KUKA KRL program: MyProgram_178().src

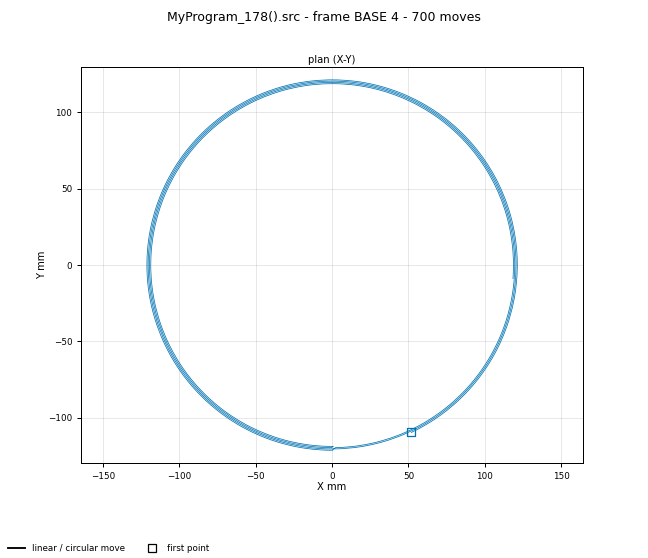
[picture p0: tool path of MyProgram_178().src in frame BASE 4, 700 of 700 moves have a stored position in this frame; points joined in program order, loops and branches not executed]
&ACCESS RVP
&REL 1
&PARAM TEMPLATE = C:\KRC\Roboter\Template\vorgabe
&PARAM EDITMASK = *
DEF MyProgram_178()
; ---- Setting reference (Base) ----
$BASE = BASE_DATA[4]

; --------------------------
; ---- Setting tool (TCP) ----
$TOOL = TOOL_DATA[3]
; --------------------------

$VEL.CP = VEL_APROX_PRINT
Startdeposition()
$VEL.CP = VEL_PRINT
LIN {X 51.9075,Y -109.6926,Z 131,A -67.6715,B 24.9586,C -1.4872,E1 25.07,E2 513.8234} C_DIS
LIN {X 55.7576,Y -107.7868,Z 131,A -65.6917,B 24.9586,C -1.4882,E1 25.0749,E2 511.8466} C_DIS
LIN {X 59.8932,Y -105.5443,Z 131,A -63.4292,B 24.9582,C -1.4942,E1 25.0805,E2 509.5764} C_DIS
LIN {X 64.6014,Y -102.7303,Z 131,A -60.7158,B 24.9576,C -1.5052,E1 25.087,E2 506.8455} C_DIS
LIN {X 68.8736,Y -99.916,Z 131,A -58.1491,B 24.9568,C -1.5177,E1 25.0929,E2 504.2581} C_DIS
LIN {X 71.8723,Y -97.7815,Z 131,A -56.8988,B 24.958,C -1.4972,E1 25.0956,E2 503.0607} C_DIS
LIN {X 75.2087,Y -95.2388,Z 131,A -54.7915,B 24.9574,C -1.5078,E1 25.1003,E2 500.9361} C_DIS
LIN {X 80.6749,Y -90.6547,Z 131,A -51.0171,B 24.9558,C -1.5358,E1 25.1084,E2 497.1104} C_DIS
LIN {X 83.659,Y -87.9089,Z 131,A -49.496,B 24.9567,C -1.5207,E1 25.1114,E2 495.631} C_DIS
LIN {X 86.4848,Y -85.1299,Z 131,A -47.1581,B 24.9551,C -1.5488,E1 25.1161,E2 493.2369} C_DIS
LIN {X 89.5631,Y -81.8851,Z 131,A -44.7373,B 24.9538,C -1.5698,E1 25.1207,E2 490.7771} C_DIS
LIN {X 93.4926,Y -77.368,Z 131,A -42.9248,B 24.9564,C -1.5263,E1 25.1238,E2 489.0757} C_DIS
LIN {X 96.0124,Y -74.2176,Z 131,A -40.5836,B 24.9548,C -1.5533,E1 25.1279,E2 486.6817} C_DIS
LIN {X 98.0547,Y -71.4981,Z 131,A -38.8834,B 24.9543,C -1.5625,E1 25.1307,E2 484.9679} C_DIS
LIN {X 100.3111,Y -68.2975,Z 131,A -37.4826,B 24.9553,C -1.5452,E1 25.1329,E2 483.6149} C_DIS
LIN {X 102.181,Y -65.4665,Z 131,A -35.8256,B 24.9548,C -1.5526,E1 25.1354,E2 481.9488} C_DIS
LIN {X 104.6437,Y -61.4536,Z 131,A -33.7099,B 24.9548,C -1.5537,E1 25.1385,E2 479.8413} C_DIS
LIN {X 106.8429,Y -57.545,Z 131,A -31.5096,B 24.9542,C -1.5641,E1 25.1414,E2 477.6278} C_DIS
LIN {X 108.0967,Y -55.1521,Z 131,A -30.1133,B 24.9536,C -1.5741,E1 25.1432,E2 476.2155} C_DIS
LIN {X 109.9322,Y -51.3961,Z 131,A -27.4409,B 24.9511,C -1.6156,E1 25.1465,E2 473.4596} C_DIS
LIN {X 112.3906,Y -45.7732,Z 131,A -25.5169,B 24.9535,C -1.5752,E1 25.1485,E2 471.6416} C_DIS
LIN {X 114.7044,Y -39.6191,Z 131,A -22.3577,B 24.9528,C -1.5877,E1 25.1515,E2 468.4705} C_DIS
LIN {X 115.9276,Y -35.8817,Z 131,A -20.6016,B 24.9528,C -1.5885,E1 25.153,E2 466.7224} C_DIS
LIN {X 118.0698,Y -28.0406,Z 131,A -16.719,B 24.9518,C -1.6031,E1 25.1558,E2 462.8278} C_DIS
LIN {X 118.8887,Y -24.3374,Z 131,A -14.9192,B 24.9515,C -1.6094,E1 25.1568,E2 461.0237} C_DIS
LIN {X 119.3717,Y -21.8423,Z 131,A -13.5562,B 24.9507,C -1.6215,E1 25.1575,E2 459.64} C_DIS
LIN {X 120.3023,Y -15.9406,Z 131,A -10.8866,B 24.9507,C -1.6231,E1 25.1586,E2 456.9824} C_DIS
LIN {X 121.1092,Y -7.7144,Z 131,A -7.2632,B 24.9507,C -1.6218,E1 25.1595,E2 453.3836} C_DIS
LIN {X 121.3487,Y -1.1842,Z 131,A -4.1632,B 24.9501,C -1.6325,E1 25.1598,E2 450.2766} C_DIS
LIN {X 121.2663,Y 4.6162,Z 131,A -0.56,B 24.9468,C -1.6853,E1 25.1595,E2 446.5706} C_DIS
LIN {X 120.9497,Y 9.8976,Z 131,A 1.0936,B 24.9489,C -1.6506,E1 25.1592,E2 445.0085} C_DIS
LIN {X 120.2667,Y 16.2062,Z 131,A 3.9191,B 24.9489,C -1.6517,E1 25.1583,E2 442.1972} C_DIS
LIN {X 119.3356,Y 22.0415,Z 131,A 6.9404,B 24.9476,C -1.6721,E1 25.1569,E2 439.1455} C_DIS
LIN {X 117.9376,Y 28.5934,Z 131,A 10.1549,B 24.9468,C -1.6846,E1 25.155,E2 435.9201} C_DIS
LIN {X 116.9158,Y 32.5181,Z 131,A 11.889,B 24.947,C -1.6815,E1 25.1537,E2 434.2033} C_DIS
LIN {X 115.8818,Y 36.0302,Z 131,A 13.7072,B 24.9464,C -1.6913,E1 25.1522,E2 432.3724} C_DIS
LIN {X 114.7061,Y 39.6143,Z 131,A 15.4665,B 24.9461,C -1.6957,E1 25.1507,E2 430.6128} C_DIS
LIN {X 113.5581,Y 42.7933,Z 131,A 18.1804,B 24.9422,C -1.7569,E1 25.1479,E2 427.7697} C_DIS
LIN {X 110.8309,Y 49.4295,Z 131,A 20.2986,B 24.9457,C -1.7028,E1 25.1457,E2 425.7906} C_DIS
LIN {X 108.6272,Y 54.1007,Z 131,A 22.8857,B 24.9447,C -1.7171,E1 25.1425,E2 423.1836} C_DIS
LIN {X 106.8006,Y 57.6239,Z 131,A 24.7746,B 24.9444,C -1.7231,E1 25.14,E2 421.2906} C_DIS
LIN {X 105.2764,Y 60.3623,Z 131,A 27.0591,B 24.9415,C -1.7674,E1 25.1367,E2 418.9133} C_DIS
LIN {X 102.1578,Y 65.5028,Z 131,A 28.9213,B 24.9442,C -1.7262,E1 25.1341,E2 417.1579} C_DIS
LIN {X 99.3296,Y 69.7163,Z 131,A 31.4724,B 24.9433,C -1.74,E1 25.13,E2 414.5866} C_DIS
LIN {X 96.7489,Y 73.2554,Z 131,A 33.5293,B 24.943,C -1.7447,E1 25.1266,E2 412.5286} C_DIS
LIN {X 94.1346,Y 76.586,Z 131,A 35.427,B 24.943,C -1.7445,E1 25.1233,E2 410.6401} C_DIS
LIN {X 91.5641,Y 79.6423,Z 131,A 37.3364,B 24.9426,C -1.7501,E1 25.1198,E2 408.7261} C_DIS
LIN {X 88.9296,Y 82.5727,Z 131,A 39.2155,B 24.9423,C -1.7553,E1 25.1163,E2 406.8432} C_DIS
LIN {X 86.0866,Y 85.5336,Z 131,A 41.1185,B 24.9421,C -1.7578,E1 25.1126,E2 404.9423} C_DIS
LIN {X 82.8873,Y 88.6374,Z 131,A 43.7663,B 24.94,C -1.789,E1 25.1071,E2 402.2319} C_DIS
LIN {X 79.4919,Y 91.6943,Z 131,A 45.3564,B 24.9416,C -1.7655,E1 25.1039,E2 400.7035} C_DIS
LIN {X 76.3668,Y 94.3129,Z 131,A 47.2601,B 24.9414,C -1.7681,E1 25.0998,E2 398.8008} C_DIS
LIN {X 73.3676,Y 96.664,Z 131,A 49.1142,B 24.941,C -1.7741,E1 25.0956,E2 396.9395} C_DIS
LIN {X 70.1538,Y 99.0214,Z 131,A 50.7217,B 24.9417,C -1.7641,E1 25.0921,E2 395.3612} C_DIS
LIN {X 65.2882,Y 102.2953,Z 131,A 53.5562,B 24.9412,C -1.7718,E1 25.0855,E2 392.5181} C_DIS
LIN {X 61.053,Y 104.8774,Z 131,A 55.9905,B 24.9406,C -1.7798,E1 25.0796,E2 390.0724} C_DIS
LIN {X 57.5811,Y 106.8236,Z 131,A 57.9333,B 24.9403,C -1.7855,E1 25.0748,E2 388.1218} C_DIS
LIN {X 54.2282,Y 108.5634,Z 131,A 59.4566,B 24.9409,C -1.7753,E1 25.0711,E2 386.6266} C_DIS
LIN {X 48.9991,Y 111.0221,Z 131,A 62.2077,B 24.9406,C -1.7796,E1 25.0642,E2 383.8723} C_DIS
LIN {X 45.1229,Y 112.6528,Z 131,A 64.3998,B 24.9398,C -1.7916,E1 25.0584,E2 381.657} C_DIS
LIN {X 41.3987,Y 114.0746,Z 131,A 66.3167,B 24.9396,C -1.795,E1 25.0534,E2 379.736} C_DIS
LIN {X 37.5457,Y 115.3998,Z 131,A 68.1965,B 24.9396,C -1.7946,E1 25.0484,E2 377.861} C_DIS
LIN {X 33.8703,Y 116.5317,Z 131,A 70.0322,B 24.9395,C -1.7969,E1 25.0435,E2 376.023} C_DIS
LIN {X 29.8443,Y 117.6272,Z 131,A 72.082,B 24.9391,C -1.8019,E1 25.0379,E2 373.9644} C_DIS
LIN {X 25.3608,Y 118.675,Z 131,A 74.6376,B 24.9378,C -1.8211,E1 25.0309,E2 371.3668} C_DIS
LIN {X 21.1845,Y 119.4906,Z 131,A 76.174,B 24.9393,C -1.7996,E1 25.0268,E2 369.8832} C_DIS
LIN {X 18.5865,Y 119.922,Z 131,A 77.7154,B 24.9383,C -1.8139,E1 25.0225,E2 368.3091} C_DIS
LIN {X 15.1404,Y 120.4056,Z 131,A 79.1736,B 24.9389,C -1.8056,E1 25.0185,E2 366.8718} C_DIS
LIN {X 9.5816,Y 120.9746,Z 131,A 81.3055,B 24.9405,C -1.7823,E1 25.0127,E2 364.7963} C_DIS
LIN {X 3.5574,Y 121.3017,Z 131,A 84.1748,B 24.9405,C -1.7831,E1 25.0047,E2 361.9261} C_DIS
LIN {X -2.1271,Y 121.3355,Z 131,A 87.1911,B 24.9394,C -1.7979,E1 24.9962,E2 358.8751} C_DIS
LIN {X -9.334,Y 120.994,Z 131,A 90.5608,B 24.9396,C -1.7949,E1 24.9868,E2 355.5116} C_DIS
LIN {X -15.8231,Y 120.3181,Z 131,A 93.4296,B 24.9404,C -1.7834,E1 24.9789,E2 352.6681} C_DIS
LIN {X -21.7635,Y 119.386,Z 131,A 96.9252,B 24.9385,C -1.8114,E1 24.9691,E2 349.1029} C_DIS
LIN {X -25.4809,Y 118.6489,Z 131,A 98.3008,B 24.9399,C -1.7909,E1 24.9655,E2 347.7743} C_DIS
LIN {X -29.1039,Y 117.8122,Z 131,A 100.1225,B 24.9398,C -1.7922,E1 24.9605,E2 345.947} C_DIS
LIN {X -33.254,Y 116.709,Z 131,A 102.1129,B 24.9401,C -1.7884,E1 24.9551,E2 343.9626} C_DIS
LIN {X -36.8342,Y 115.6286,Z 131,A 103.711,B 24.9407,C -1.7788,E1 24.9509,E2 342.3845} C_DIS
LIN {X -42.7165,Y 113.5872,Z 131,A 106.8783,B 24.9403,C -1.7852,E1 24.9425,E2 339.1956} C_DIS
LIN {X -46.3503,Y 112.1535,Z 131,A 108.674,B 24.9406,C -1.7804,E1 24.9379,E2 337.4073} C_DIS
LIN {X -49.6007,Y 110.7549,Z 131,A 110.421,B 24.9406,C -1.7814,E1 24.9334,E2 335.654} C_DIS
LIN {X -53.6807,Y 108.8359,Z 131,A 112.5091,B 24.9409,C -1.7761,E1 24.9282,E2 333.5729} C_DIS
LIN {X -57.1689,Y 107.0442,Z 131,A 114.1462,B 24.9417,C -1.7635,E1 24.9242,E2 331.9614} C_DIS
LIN {X -61.8681,Y 104.3984,Z 131,A 116.9551,B 24.9412,C -1.7706,E1 24.9173,E2 329.1273} C_DIS
LIN {X -66.4465,Y 101.5464,Z 131,A 119.4941,B 24.9416,C -1.7653,E1 24.9114,E2 326.5928} C_DIS
LIN {X -69.7163,Y 99.3296,Z 131,A 121.4321,B 24.9416,C -1.7648,E1 24.9069,E2 324.6495} C_DIS
LIN {X -75.213,Y 95.2349,Z 131,A 124.9477,B 24.9413,C -1.7702,E1 24.899,E2 321.1081} C_DIS
LIN {X -78.0269,Y 92.9448,Z 131,A 126.3432,B 24.9425,C -1.7523,E1 24.8961,E2 319.75} C_DIS
LIN {X -79.9811,Y 91.2675,Z 131,A 127.8598,B 24.9418,C -1.7628,E1 24.8929,E2 318.2025} C_DIS
LIN {X -82.5152,Y 88.9831,Z 131,A 129.6047,B 24.9416,C -1.7649,E1 24.8893,E2 316.4454} C_DIS
LIN {X -85.4186,Y 86.2004,Z 131,A 131.1002,B 24.9431,C -1.7425,E1 24.8864,E2 314.997} C_DIS
LIN {X -88.6122,Y 82.9141,Z 131,A 133.5621,B 24.9426,C -1.7502,E1 24.8816,E2 312.5061} C_DIS
LIN {X -90.8963,Y 80.4034,Z 131,A 135.1198,B 24.943,C -1.7441,E1 24.8787,E2 310.9559} C_DIS
LIN {X -95.0583,Y 75.4372,Z 131,A 137.9487,B 24.9442,C -1.7258,E1 24.8738,E2 308.1573} C_DIS
LIN {X -97.8995,Y 71.7111,Z 131,A 140.1737,B 24.9445,C -1.7203,E1 24.8701,E2 305.9348} C_DIS
LIN {X -101.4777,Y 66.5508,Z 131,A 143.0393,B 24.9454,C -1.7077,E1 24.8656,E2 303.0851} C_DIS
LIN {X -104.0799,Y 62.4035,Z 131,A 145.4404,B 24.9455,C -1.7048,E1 24.8621,E2 300.6785} C_DIS
LIN {X -107.1965,Y 56.8833,Z 131,A 148.5248,B 24.9458,C -1.6999,E1 24.8579,E2 297.5895} C_DIS
LIN {X -109.1931,Y 52.9505,Z 131,A 151.4913,B 24.9438,C -1.7323,E1 24.8542,E2 294.5298} C_DIS
LIN {X -111.738,Y 47.3419,Z 131,A 153.4814,B 24.9469,C -1.6832,E1 24.8521,E2 292.6458} C_DIS
LIN {X -113.2889,Y 43.5024,Z 131,A 155.5141,B 24.9471,C -1.6805,E1 24.85,E2 290.6083} C_DIS
LIN {X -115.1337,Y 38.3549,Z 131,A 158.1108,B 24.9476,C -1.6729,E1 24.8476,E2 288.0147} C_DIS
LIN {X -116.4113,Y 34.2806,Z 131,A 159.9049,B 24.9486,C -1.657,E1 24.8461,E2 286.2484} C_DIS
LIN {X -118.1334,Y 27.7741,Z 131,A 163.3441,B 24.9485,C -1.6579,E1 24.8437,E2 282.7868} C_DIS
LIN {X -118.9425,Y 24.0726,Z 131,A 165.0375,B 24.9491,C -1.648,E1 24.8428,E2 281.1072} C_DIS
LIN {X -119.6198,Y 20.4409,Z 131,A 166.9038,B 24.9491,C -1.6476,E1 24.8418,E2 279.2307} C_DIS
LIN {X -120.179,Y 16.8455,Z 131,A 168.6443,B 24.9494,C -1.643,E1 24.8411,E2 277.4909} C_DIS
LIN {X -120.7282,Y 12.3096,Z 131,A 171.0854,B 24.9491,C -1.6482,E1 24.8404,E2 275.0226} C_DIS
LIN {X -121.0302,Y 8.8657,Z 131,A 172.4566,B 24.9501,C -1.6315,E1 24.8401,E2 273.6829} C_DIS
LIN {X -121.2587,Y 4.7995,Z 131,A 174.2869,B 24.9507,C -1.6212,E1 24.8399,E2 271.8662} C_DIS
LIN {X -121.3508,Y 0.8369,Z 131,A 176.1792,B 24.9511,C -1.616,E1 24.8398,E2 269.9749} C_DIS
LIN {X -121.343,Y -1.6133,Z 131,A 177.5598,B 24.9507,C -1.6219,E1 24.8398,E2 268.5719} C_DIS
LIN {X -121.1399,Y -7.2007,Z 131,A -179.8825,B 24.9514,C -1.6098,E1 24.8402,E2 266.0278} C_DIS
LIN {X -120.836,Y -11.2024,Z 131,A -177.9847,B 24.9518,C -1.6037,E1 24.8406,E2 264.133} C_DIS
LIN {X -120.3784,Y -15.359,Z 131,A -176.0064,B 24.9522,C -1.5975,E1 24.8413,E2 262.1577} C_DIS
LIN {X -119.8144,Y -19.268,Z 131,A -174.2451,B 24.9528,C -1.5871,E1 24.842,E2 260.4107} C_DIS
LIN {X -119.1451,Y -23.048,Z 131,A -172.3772,B 24.953,C -1.5838,E1 24.843,E2 258.5397} C_DIS
LIN {X -118.3394,Y -26.8795,Z 131,A -170.4695,B 24.9532,C -1.5805,E1 24.8441,E2 256.6286} C_DIS
LIN {X -117.353,Y -30.9064,Z 131,A -167.8257,B 24.9518,C -1.6044,E1 24.846,E2 253.9123} C_DIS
LIN {X -115.9462,Y -35.8212,Z 131,A -166.0638,B 24.9539,C -1.5685,E1 24.8474,E2 252.226} C_DIS
LIN {X -114.6294,Y -39.8345,Z 131,A -164.2266,B 24.9547,C -1.5556,E1 24.849,E2 250.4091} C_DIS
LIN {X -112.0973,Y -46.4867,Z 131,A -160.6042,B 24.9546,C -1.5569,E1 24.8527,E2 246.7631} C_DIS
LIN {X -110.2477,Y -50.7188,Z 131,A -158.4108,B 24.9549,C -1.5512,E1 24.8552,E2 244.5714} C_DIS
LIN {X -108.2864,Y -54.781,Z 131,A -156.4727,B 24.9558,C -1.5367,E1 24.8576,E2 242.6572} C_DIS
LIN {X -105.3435,Y -60.2448,Z 131,A -153.3965,B 24.9558,C -1.535,E1 24.8617,E2 239.5689} C_DIS
LIN {X -103.2114,Y -63.8291,Z 131,A -151.4088,B 24.9561,C -1.5306,E1 24.8646,E2 237.5816} C_DIS
LIN {X -101.7362,Y -66.1554,Z 131,A -150.0444,B 24.9561,C -1.53,E1 24.8667,E2 236.2117} C_DIS
LIN {X -99.3673,Y -69.6623,Z 131,A -148.0547,B 24.9565,C -1.5245,E1 24.8698,E2 234.2254} C_DIS
LIN {X -97.122,Y -72.761,Z 131,A -145.7555,B 24.9555,C -1.5419,E1 24.8738,E2 231.8736} C_DIS
LIN {X -94.3764,Y -76.2884,Z 131,A -144.1459,B 24.957,C -1.5144,E1 24.8765,E2 230.3219} C_DIS
LIN {X -91.7091,Y -79.4747,Z 131,A -142.4479,B 24.958,C -1.4981,E1 24.8795,E2 228.6549} C_DIS
LIN {X -88.2916,Y -83.2546,Z 131,A -139.783,B 24.9576,C -1.5041,E1 24.8845,E2 225.9639} C_DIS
LIN {X -82.8742,Y -88.6495,Z 131,A -136.0908,B 24.9578,C -1.5001,E1 24.8919,E2 222.2658} C_DIS
LIN {X -79.7679,Y -91.4544,Z 131,A -134.1365,B 24.9581,C -1.4952,E1 24.896,E2 220.3155} C_DIS
LIN {X -76.5396,Y -94.1724,Z 131,A -132.1226,B 24.9583,C -1.4923,E1 24.9003,E2 218.3007} C_DIS
LIN {X -72.9252,Y -96.9986,Z 131,A -129.4317,B 24.9572,C -1.5122,E1 24.9064,E2 215.5527} C_DIS
LIN {X -69.1991,Y -99.691,Z 131,A -127.7818,B 24.9587,C -1.4849,E1 24.9101,E2 213.9623} C_DIS
LIN {X -65.6529,Y -102.0612,Z 131,A -125.582,B 24.9584,C -1.4901,E1 24.9153,E2 211.7429} C_DIS
LIN {X -61.7558,Y -104.4655,Z 131,A -123.5906,B 24.959,C -1.4791,E1 24.92,E2 209.7715} C_DIS
LIN {X -58.0803,Y -106.5525,Z 131,A -121.6067,B 24.9592,C -1.4758,E1 24.9248,E2 207.7898} C_DIS
LIN {X -52.2099,Y -109.5482,Z 131,A -118.4902,B 24.9594,C -1.472,E1 24.9326,E2 204.6739} C_DIS
LIN {X -47.3662,Y -111.7278,Z 131,A -116.0212,B 24.9597,C -1.4675,E1 24.9389,E2 202.2098} C_DIS
LIN {X -43.7519,Y -113.1928,Z 131,A -114.1366,B 24.9597,C -1.4676,E1 24.9438,E2 200.3208} C_DIS
LIN {X -40.1344,Y -114.5249,Z 131,A -112.3526,B 24.9598,C -1.4644,E1 24.9485,E2 198.5409} C_DIS
LIN {X -36.4443,Y -115.7525,Z 131,A -110.4578,B 24.9598,C -1.4656,E1 24.9535,E2 196.6397} C_DIS
LIN {X -32.6677,Y -116.8742,Z 131,A -108.4402,B 24.9594,C -1.4717,E1 24.959,E2 194.6046} C_DIS
LIN {X -28.4607,Y -117.9695,Z 131,A -106.0229,B 24.9585,C -1.4876,E1 24.9657,E2 192.146} C_DIS
LIN {X -24.0711,Y -118.9427,Z 131,A -104.535,B 24.9602,C -1.4569,E1 24.9695,E2 190.7293} C_DIS
LIN {X -21.2873,Y -119.4721,Z 131,A -102.9586,B 24.9597,C -1.4676,E1 24.9739,E2 189.1259} C_DIS
LIN {X -17.8075,Y -120.0409,Z 131,A -101.1844,B 24.9594,C -1.4723,E1 24.9789,E2 187.339} C_DIS
LIN {X -12.7375,Y -120.6831,Z 131,A -99.2145,B 24.9606,C -1.4511,E1 24.9842,E2 185.4181} C_DIS
LIN {X -7.453,Y -121.1248,Z 131,A -96.0396,B 24.9588,C -1.4828,E1 24.9933,E2 182.1667} C_DIS
LIN {X -3.2189,Y -121.3118,Z 131,A -94.4845,B 24.96,C -1.4618,E1 24.9975,E2 180.6612} C_DIS
LIN {X 0.4041,Y -121.3528,Z 131,A -92.2335,B 24.9585,C -1.488,E1 25.0039,E2 178.3481} C_DIS
LIN {X 0.4041,Y -121.3528,Z 131,A -92.2335,B 24.9585,C -1.488,E1 25.0039,E2 178.3481} C_DIS
Enddeposition()
LIN {X 0.8351,Y -120.4889,Z 131,A -92.1393,B 24.958,C -1.4976,E1 25.0042,E2 178.2313} C_DIS
Startdeposition()
$VEL.CP = VEL_PRINT
LIN {X -3.9171,Y -120.4489,Z 131,A -95.8339,B 24.9617,C -1.4296,E1 24.9935,E2 182.0872} C_DIS
LIN {X -9.0404,Y -120.1728,Z 131,A -98.3701,B 24.962,C -1.4251,E1 24.9864,E2 184.635} C_DIS
LIN {X -13.0956,Y -119.7998,Z 131,A -100.5414,B 24.9625,C -1.4145,E1 24.9803,E2 186.8325} C_DIS
LIN {X -17.0407,Y -119.3019,Z 131,A -101.8416,B 24.9611,C -1.4419,E1 24.9769,E2 188.0689} C_DIS
LIN {X -19.7696,Y -118.881,Z 131,A -103.235,B 24.9612,C -1.4386,E1 24.973,E2 189.4714} C_DIS
LIN {X -22.9331,Y -118.3111,Z 131,A -104.8232,B 24.9613,C -1.4364,E1 24.9686,E2 191.0664} C_DIS
LIN {X -27.6575,Y -117.2967,Z 131,A -107.109,B 24.9613,C -1.438,E1 24.9624,E2 193.3512} C_DIS
LIN {X -31.9009,Y -116.2148,Z 131,A -109.2087,B 24.9613,C -1.4385,E1 24.9567,E2 195.4529} C_DIS
LIN {X -35.7931,Y -115.0752,Z 131,A -111.1624,B 24.9613,C -1.4387,E1 24.9515,E2 197.4094} C_DIS
LIN {X -39.5661,Y -113.8327,Z 131,A -113.041,B 24.9611,C -1.4408,E1 24.9465,E2 199.2867} C_DIS
LIN {X -43.4461,Y -112.4097,Z 131,A -115.0192,B 24.9611,C -1.442,E1 24.9413,E2 201.2661} C_DIS
LIN {X -47.9767,Y -110.5513,Z 131,A -117.2877,B 24.9608,C -1.4471,E1 24.9355,E2 203.5276} C_DIS
LIN {X -51.391,Y -109.007,Z 131,A -119.1366,B 24.9608,C -1.4462,E1 24.9308,E2 205.3833} C_DIS
LIN {X -55.7885,Y -106.8224,Z 131,A -121.2371,B 24.9601,C -1.4596,E1 24.9256,E2 207.4575} C_DIS
LIN {X -58.2872,Y -105.4809,Z 131,A -122.8699,B 24.9607,C -1.4487,E1 24.9216,E2 209.1208} C_DIS
LIN {X -61.7284,Y -103.5036,Z 131,A -124.8047,B 24.9607,C -1.4494,E1 24.9169,E2 211.0599} C_DIS
LIN {X -65.0323,Y -101.4609,Z 131,A -126.6452,B 24.9605,C -1.4525,E1 24.9125,E2 212.8988} C_DIS
LIN {X -68.846,Y -98.9127,Z 131,A -128.6931,B 24.96,C -1.462,E1 24.9079,E2 214.9311} C_DIS
LIN {X -72.8208,Y -96.0236,Z 131,A -131.0965,B 24.9599,C -1.4631,E1 24.9024,E2 217.3403} C_DIS
LIN {X -75.9695,Y -93.5526,Z 131,A -133.0353,B 24.9598,C -1.4651,E1 24.8982,E2 219.2816} C_DIS
LIN {X -79.2342,Y -90.8043,Z 131,A -135.0464,B 24.9595,C -1.4699,E1 24.8939,E2 221.2892} C_DIS
LIN {X -82.198,Y -88.1303,Z 131,A -137.7144,B 24.9611,C -1.4404,E1 24.8883,E2 224.0383} C_DIS
LIN {X -86.1006,Y -84.3213,Z 131,A -139.4107,B 24.9587,C -1.4848,E1 24.8852,E2 225.6361} C_DIS
LIN {X -90.0357,Y -80.1061,Z 131,A -142.1412,B 24.9583,C -1.4914,E1 24.88,E2 228.3628} C_DIS
LIN {X -92.2217,Y -77.5803,Z 131,A -143.9402,B 24.9586,C -1.4859,E1 24.8767,E2 230.183} C_DIS
LIN {X -95.7174,Y -73.2221,Z 131,A -146.684,B 24.9585,C -1.4886,E1 24.8719,E2 232.9333} C_DIS
LIN {X -97.706,Y -70.5487,Z 131,A -148.2233,B 24.9582,C -1.4945,E1 24.8694,E2 234.4661} C_DIS
LIN {X -100.4994,Y -66.507,Z 131,A -150.4741,B 24.9576,C -1.5042,E1 24.8659,E2 236.705} C_DIS
LIN {X -102.5149,Y -63.3572,Z 131,A -152.309,B 24.9575,C -1.5065,E1 24.8632,E2 238.5438} C_DIS
LIN {X -104.4826,Y -60.057,Z 131,A -154.1314,B 24.9572,C -1.5116,E1 24.8606,E2 240.3634} C_DIS
LIN {X -107.0555,Y -55.3412,Z 131,A -156.5082,B 24.9564,C -1.5263,E1 24.8575,E2 242.7178} C_DIS
LIN {X -109.1051,Y -51.1806,Z 131,A -158.9217,B 24.9565,C -1.5236,E1 24.8545,E2 245.1507} C_DIS
LIN {X -110.7091,Y -47.6124,Z 131,A -160.8195,B 24.9563,C -1.5274,E1 24.8524,E2 247.0499} C_DIS
LIN {X -113.9154,Y -39.3287,Z 131,A -164.9098,B 24.9552,C -1.5456,E1 24.8484,E2 251.1199} C_DIS
LIN {X -114.8659,Y -36.4587,Z 131,A -167.3752,B 24.9575,C -1.5067,E1 24.8462,E2 253.6923} C_DIS
LIN {X -116.5381,Y -30.6997,Z 131,A -169.4337,B 24.9551,C -1.5487,E1 24.8447,E2 255.6625} C_DIS
LIN {X -117.5227,Y -26.6796,Z 131,A -171.4023,B 24.9547,C -1.5549,E1 24.8435,E2 257.628} C_DIS
LIN {X -118.376,Y -22.5936,Z 131,A -173.3196,B 24.9542,C -1.564,E1 24.8424,E2 259.5349} C_DIS
LIN {X -119.0555,Y -18.6893,Z 131,A -175.2559,B 24.9539,C -1.5678,E1 24.8415,E2 261.4737} C_DIS
LIN {X -119.6059,Y -14.7595,Z 131,A -177.1972,B 24.9537,C -1.5716,E1 24.8408,E2 263.4175} C_DIS
LIN {X -120.047,Y -10.5893,Z 131,A -179.1451,B 24.9532,C -1.5799,E1 24.8403,E2 265.3572} C_DIS
LIN {X -120.3191,Y -6.8438,Z 131,A 178.9314,B 24.9532,C -1.5799,E1 24.84,E2 267.2922} C_DIS
LIN {X -120.4882,Y -2.4665,Z 131,A 176.9449,B 24.9526,C -1.5907,E1 24.8398,E2 269.2649} C_DIS
LIN {X -120.5052,Y 1.4021,Z 131,A 175.0535,B 24.9524,C -1.5946,E1 24.8398,E2 271.1587} C_DIS
LIN {X -120.3971,Y 5.2875,Z 131,A 173.2349,B 24.9519,C -1.6019,E1 24.84,E2 272.9707} C_DIS
LIN {X -120.1709,Y 9.0777,Z 131,A 171.1758,B 24.9522,C -1.5971,E1 24.8404,E2 275.0535} C_DIS
LIN {X -119.6855,Y 14.0997,Z 131,A 168.9757,B 24.9512,C -1.6133,E1 24.8411,E2 277.2283} C_DIS
LIN {X -119.1614,Y 17.9985,Z 131,A 167.1606,B 24.9507,C -1.6217,E1 24.8418,E2 279.0341} C_DIS
LIN {X -118.542,Y 21.7064,Z 131,A 165.2879,B 24.9506,C -1.624,E1 24.8427,E2 280.9126} C_DIS
LIN {X -117.809,Y 25.3869,Z 131,A 163.5334,B 24.9502,C -1.631,E1 24.8437,E2 282.6607} C_DIS
LIN {X -115.9261,Y 32.933,Z 131,A 159.8097,B 24.9495,C -1.6417,E1 24.8463,E2 286.3804} C_DIS
LIN {X -114.7622,Y 36.7848,Z 131,A 157.5301,B 24.9501,C -1.6324,E1 24.8482,E2 288.6953} C_DIS
LIN {X -113.6445,Y 40.1051,Z 131,A 156.2837,B 24.9487,C -1.6553,E1 24.8493,E2 289.8943} C_DIS
LIN {X -112.4635,Y 43.308,Z 131,A 154.5143,B 24.9487,C -1.6542,E1 24.851,E2 291.6763} C_DIS
LIN {X -110.9107,Y 47.1402,Z 131,A 152.1136,B 24.9495,C -1.6421,E1 24.8537,E2 294.1193} C_DIS
LIN {X -109.2556,Y 50.8578,Z 131,A 150.1386,B 24.9492,C -1.6463,E1 24.856,E2 296.095} C_DIS
LIN {X -107.404,Y 54.6603,Z 131,A 147.5982,B 24.9502,C -1.6303,E1 24.8593,E2 298.6871} C_DIS
LIN {X -104.2409,Y 60.4759,Z 131,A 145.6548,B 24.9465,C -1.69,E1 24.8618,E2 300.4983} C_DIS
LIN {X -102.8639,Y 62.7881,Z 131,A 144.0936,B 24.947,C -1.6818,E1 24.8641,E2 302.0871} C_DIS
LIN {X -100.8552,Y 65.9677,Z 131,A 141.6941,B 24.9483,C -1.6611,E1 24.8679,E2 304.548} C_DIS
LIN {X -98.0665,Y 70.0446,Z 131,A 139.6496,B 24.9471,C -1.6804,E1 24.8711,E2 306.5565} C_DIS
LIN {X -95.9567,Y 72.9093,Z 131,A 138.5747,B 24.9451,C -1.7112,E1 24.8728,E2 307.5632} C_DIS
LIN {X -92.8884,Y 76.7797,Z 131,A 135.941,B 24.9455,C -1.7053,E1 24.8774,E2 310.2233} C_DIS
LIN {X -90.3146,Y 79.7919,Z 131,A 133.9728,B 24.9455,C -1.7066,E1 24.881,E2 312.1973} C_DIS
LIN {X -87.1791,Y 83.2071,Z 131,A 131.7483,B 24.9451,C -1.7113,E1 24.8853,E2 314.4204} C_DIS
LIN {X -84.0995,Y 86.3184,Z 131,A 129.4912,B 24.9453,C -1.7089,E1 24.8898,E2 316.6928} C_DIS
LIN {X -80.2604,Y 89.8976,Z 131,A 127.2689,B 24.9441,C -1.7264,E1 24.8943,E2 318.8822} C_DIS
LIN {X -77.2783,Y 92.474,Z 131,A 124.7163,B 24.9457,C -1.7017,E1 24.8999,E2 321.5037} C_DIS
LIN {X -73.5556,Y 95.4613,Z 131,A 123.0655,B 24.9437,C -1.733,E1 24.9034,E2 323.0858} C_DIS
LIN {X -70.9623,Y 97.4049,Z 131,A 121.5845,B 24.9433,C -1.7388,E1 24.9067,E2 324.5582} C_DIS
LIN {X -67.7964,Y 99.6353,Z 131,A 119.6499,B 24.9433,C -1.7385,E1 24.9111,E2 326.5003} C_DIS
LIN {X -64.0987,Y 102.0534,Z 131,A 117.76,B 24.9425,C -1.7517,E1 24.9155,E2 328.3648} C_DIS
LIN {X -59.7783,Y 104.6419,Z 131,A 114.9797,B 24.9433,C -1.7393,E1 24.9223,E2 331.1829} C_DIS
LIN {X -55.4128,Y 107.0187,Z 131,A 112.6769,B 24.9429,C -1.746,E1 24.928,E2 333.4764} C_DIS
LIN {X -51.9039,Y 108.7628,Z 131,A 110.9927,B 24.9422,C -1.7568,E1 24.9321,E2 335.1392} C_DIS
LIN {X -48.8591,Y 110.1644,Z 131,A 109.3451,B 24.9422,C -1.7568,E1 24.9363,E2 336.7908} C_DIS
LIN {X -45.6112,Y 111.5486,Z 131,A 107.6516,B 24.942,C -1.7586,E1 24.9407,E2 338.4839} C_DIS
LIN {X -41.9847,Y 112.9635,Z 131,A 105.189,B 24.9436,C -1.7344,E1 24.9473,E2 341.0093} C_DIS
LIN {X -37.658,Y 114.4783,Z 131,A 103.9093,B 24.9408,C -1.7765,E1 24.9504,E2 342.1912} C_DIS
LIN {X -34.9893,Y 115.3227,Z 131,A 102.1857,B 24.9419,C -1.7607,E1 24.9551,E2 343.9555} C_DIS
LIN {X -30.862,Y 116.4946,Z 131,A 100.2066,B 24.9416,C -1.7655,E1 24.9604,E2 345.9261} C_DIS
LIN {X -27.2005,Y 117.4034,Z 131,A 98.3979,B 24.9416,C -1.7666,E1 24.9653,E2 347.7348} C_DIS
LIN {X -19.0968,Y 118.9906,Z 131,A 94.7891,B 24.9404,C -1.7838,E1 24.9752,E2 351.3065} C_DIS
LIN {X -14.8331,Y 119.5968,Z 131,A 91.902,B 24.9428,C -1.7477,E1 24.9834,E2 354.2816} C_DIS
LIN {X -10.5267,Y 120.0524,Z 131,A 90.478,B 24.9408,C -1.777,E1 24.9871,E2 355.6367} C_DIS
LIN {X -4.7406,Y 120.4198,Z 131,A 87.9671,B 24.94,C -1.7892,E1 24.9941,E2 358.1197} C_DIS
LIN {X 1.9366,Y 120.4975,Z 131,A 84.5108,B 24.9408,C -1.7771,E1 25.0038,E2 361.6046} C_DIS
LIN {X 6.4779,Y 120.3394,Z 131,A 82.4949,B 24.9404,C -1.7838,E1 25.0094,E2 363.6041} C_DIS
LIN {X 9.3197,Y 120.1519,Z 131,A 80.4771,B 24.9424,C -1.7536,E1 25.0152,E2 365.6924} C_DIS
LIN {X 13.2559,Y 119.7819,Z 131,A 78.8489,B 24.9416,C -1.7647,E1 25.0196,E2 367.2933} C_DIS
LIN {X 17.8249,Y 119.1879,Z 131,A 76.7951,B 24.9413,C -1.7703,E1 25.0253,E2 369.3318} C_DIS
LIN {X 22.0183,Y 118.4855,Z 131,A 74.6486,B 24.9417,C -1.7639,E1 25.0312,E2 371.4914} C_DIS
LIN {X 25.547,Y 117.7741,Z 131,A 73.1249,B 24.9412,C -1.7716,E1 25.0353,E2 372.9947} C_DIS
LIN {X 29.0505,Y 116.9592,Z 131,A 71.4973,B 24.941,C -1.7745,E1 25.0397,E2 374.6133} C_DIS
LIN {X 32.6525,Y 116.0059,Z 131,A 69.5957,B 24.9415,C -1.7673,E1 25.0449,E2 376.5289} C_DIS
LIN {X 36.4848,Y 114.8576,Z 131,A 67.7073,B 24.9415,C -1.7664,E1 25.0499,E2 378.4158} C_DIS
LIN {X 40.3452,Y 113.5597,Z 131,A 65.7373,B 24.9417,C -1.7632,E1 25.0551,E2 380.3897} C_DIS
LIN {X 45.6776,Y 111.5212,Z 131,A 63.4193,B 24.9407,C -1.7789,E1 25.061,E2 382.6654} C_DIS
LIN {X 49.8214,Y 109.7325,Z 131,A 60.5979,B 24.9429,C -1.7449,E1 25.0684,E2 385.5602} C_DIS
LIN {X 53.0655,Y 108.2011,Z 131,A 59.4457,B 24.9414,C -1.7686,E1 25.0712,E2 386.6533} C_DIS
LIN {X 55.678,Y 106.8802,Z 131,A 57.8644,B 24.9421,C -1.7579,E1 25.0752,E2 388.2556} C_DIS
LIN {X 59.2365,Y 104.9503,Z 131,A 55.6555,B 24.9431,C -1.7419,E1 25.0806,E2 390.496} C_DIS
LIN {X 62.0711,Y 103.2992,Z 131,A 54.556,B 24.9419,C -1.7612,E1 25.0832,E2 391.5465} C_DIS
LIN {X 64.7566,Y 101.6369,Z 131,A 52.8826,B 24.9426,C -1.7507,E1 25.0872,E2 393.2393} C_DIS
LIN {X 69.1571,Y 98.6949,Z 131,A 50.3691,B 24.9428,C -1.7466,E1 25.093,E2 395.7539} C_DIS
LIN {X 72.4469,Y 96.3064,Z 131,A 48.4217,B 24.9431,C -1.7425,E1 25.0973,E2 397.7041} C_DIS
LIN {X 75.6525,Y 93.8098,Z 131,A 46.5111,B 24.9433,C -1.7399,E1 25.1015,E2 399.6138} C_DIS
LIN {X 78.7182,Y 91.2516,Z 131,A 44.3094,B 24.9444,C -1.7217,E1 25.1063,E2 401.8498} C_DIS
LIN {X 81.328,Y 88.9334,Z 131,A 42.812,B 24.9442,C -1.726,E1 25.1093,E2 403.331} C_DIS
LIN {X 84.7547,Y 85.6745,Z 131,A 40.7277,B 24.944,C -1.729,E1 25.1135,E2 405.3995} C_DIS
LIN {X 87.6514,Y 82.7082,Z 131,A 38.787,B 24.9442,C -1.7261,E1 25.1172,E2 407.3386} C_DIS
LIN {X 90.4283,Y 79.6625,Z 131,A 36.823,B 24.9445,C -1.7214,E1 25.1209,E2 409.305} C_DIS
LIN {X 93.1587,Y 76.4523,Z 131,A 34.8025,B 24.9448,C -1.7158,E1 25.1245,E2 411.3295} C_DIS
LIN {X 95.7791,Y 73.1433,Z 131,A 32.8267,B 24.945,C -1.7124,E1 25.1279,E2 413.3041} C_DIS
LIN {X 98.1227,Y 69.9659,Z 131,A 30.7959,B 24.9458,C -1.7002,E1 25.1313,E2 415.3537} C_DIS
LIN {X 100.102,Y 67.1045,Z 131,A 29.2872,B 24.9457,C -1.7029,E1 25.1336,E2 416.8486} C_DIS
LIN {X 102.3258,Y 63.6616,Z 131,A 26.9102,B 24.9473,C -1.6771,E1 25.1372,E2 419.2744} C_DIS
LIN {X 104.5064,Y 60.0153,Z 131,A 25.6874,B 24.9452,C -1.7102,E1 25.1388,E2 420.4129} C_DIS
LIN {X 105.8082,Y 57.6892,Z 131,A 24.1476,B 24.9463,C -1.6934,E1 25.1409,E2 421.9843} C_DIS
LIN {X 107.5964,Y 54.2823,Z 131,A 22.0765,B 24.9473,C -1.6765,E1 25.1436,E2 424.0844} C_DIS
LIN {X 109.4267,Y 50.4907,Z 131,A 20.344,B 24.9469,C -1.6838,E1 25.1456,E2 425.7902} C_DIS
LIN {X 110.977,Y 46.9831,Z 131,A 17.8171,B 24.9493,C -1.6444,E1 25.1485,E2 428.3962} C_DIS
LIN {X 112.9159,Y 42.1136,Z 131,A 16.2777,B 24.9469,C -1.6832,E1 25.1499,E2 429.8355} C_DIS
LIN {X 114.3627,Y 38.0103,Z 131,A 13.9178,B 24.9482,C -1.6627,E1 25.1521,E2 432.2305} C_DIS
LIN {X 115.577,Y 34.1368,Z 131,A 12.0541,B 24.9484,C -1.66,E1 25.1536,E2 434.0899} C_DIS
LIN {X 116.6196,Y 30.3852,Z 131,A 10.2171,B 24.9487,C -1.655,E1 25.155,E2 435.9282} C_DIS
LIN {X 117.8886,Y 25.0152,Z 131,A 7.5752,B 24.9492,C -1.6458,E1 25.1566,E2 438.5765} C_DIS
LIN {X 118.6903,Y 20.885,Z 131,A 5.323,B 24.9504,C -1.6271,E1 25.1577,E2 440.8596} C_DIS
LIN {X 119.2263,Y 17.5667,Z 131,A 3.369,B 24.9518,C -1.6046,E1 25.1585,E2 442.8551} C_DIS
LIN {X 119.8598,Y 12.5291,Z 131,A 1.6382,B 24.9502,C -1.6302,E1 25.1591,E2 444.5153} C_DIS
LIN {X 120.3773,Y 5.731,Z 131,A -1.3987,B 24.9502,C -1.6297,E1 25.1597,E2 447.5353} C_DIS
LIN {X 120.5094,Y 0.9637,Z 131,A -3.8628,B 24.9513,C -1.6126,E1 25.1597,E2 450.0251} C_DIS
LIN {X 120.3329,Y -6.5955,Z 131,A -7.1585,B 24.9511,C -1.6155,E1 25.1595,E2 453.2942} C_DIS
LIN {X 119.8404,Y -12.7126,Z 131,A -10.1902,B 24.952,C -1.6003,E1 25.1588,E2 456.3439} C_DIS
LIN {X 119.0853,Y -18.4963,Z 131,A -13.0424,B 24.9528,C -1.5873,E1 25.1577,E2 459.21} C_DIS
LIN {X 118.4542,Y -22.1829,Z 131,A -14.7787,B 24.953,C -1.5835,E1 25.1569,E2 460.9449} C_DIS
LIN {X 117.7221,Y -25.7841,Z 131,A -16.4931,B 24.9533,C -1.5795,E1 25.1559,E2 462.6589} C_DIS
LIN {X 116.931,Y -29.164,Z 131,A -18.6278,B 24.955,C -1.5503,E1 25.1544,E2 464.85} C_DIS
LIN {X 115.8923,Y -33.0523,Z 131,A -20.0793,B 24.954,C -1.5668,E1 25.1534,E2 466.2542} C_DIS
LIN {X 114.7983,Y -36.6714,Z 131,A -21.9068,B 24.9544,C -1.5596,E1 25.1518,E2 468.0884} C_DIS
LIN {X 112.9017,Y -42.1519,Z 131,A -24.6853,B 24.955,C -1.5498,E1 25.1492,E2 470.8743} C_DIS
LIN {X 111.4384,Y -45.879,Z 131,A -26.4209,B 24.9549,C -1.5522,E1 25.1474,E2 472.5947} C_DIS
LIN {X 109.1087,Y -51.1729,Z 131,A -29.2199,B 24.9555,C -1.5413,E1 25.1442,E2 475.4042} C_DIS
LIN {X 107.2651,Y -54.9318,Z 131,A -31.1936,B 24.9558,C -1.5361,E1 25.1418,E2 477.3797} C_DIS
LIN {X 104.822,Y -59.4629,Z 131,A -33.4565,B 24.9557,C -1.5379,E1 25.1388,E2 479.6265} C_DIS
LIN {X 103.495,Y -61.7428,Z 131,A -34.9741,B 24.9566,C -1.5212,E1 25.1366,E2 481.1756} C_DIS
LIN {X 101.8592,Y -64.406,Z 131,A -36.3145,B 24.9565,C -1.524,E1 25.1346,E2 482.5026} C_DIS
LIN {X 99.9707,Y -67.2994,Z 131,A -37.9336,B 24.9567,C -1.5205,E1 25.1321,E2 484.122} C_DIS
LIN {X 97.4895,Y -70.8461,Z 131,A -40.6949,B 24.9589,C -1.4805,E1 25.1275,E2 486.9642} C_DIS
LIN {X 94.4657,Y -74.8313,Z 131,A -42.4096,B 24.9575,C -1.5063,E1 25.1246,E2 488.6101} C_DIS
LIN {X 89.9768,Y -80.1719,Z 131,A -45.4209,B 24.9571,C -1.5124,E1 25.1193,E2 491.5931} C_DIS
LIN {X 85.434,Y -84.9973,Z 131,A -48.5626,B 24.9576,C -1.5048,E1 25.1132,E2 494.739} C_DIS
LIN {X 80.7012,Y -89.5029,Z 131,A -52.02,B 24.959,C -1.4802,E1 25.1061,E2 498.2405} C_DIS
LIN {X 77.069,Y -92.648,Z 131,A -54.1112,B 24.9587,C -1.4843,E1 25.1017,E2 500.3138} C_DIS
LIN {X 71.8978,Y -96.7167,Z 131,A -57.4538,B 24.9597,C -1.4671,E1 25.0942,E2 503.6848} C_DIS
LIN {X 67.9826,Y -99.5081,Z 131,A -59.6757,B 24.9597,C -1.4654,E1 25.0892,E2 505.9029} C_DIS
LIN {X 62.6301,Y -102.96,Z 131,A -62.5345,B 24.9597,C -1.4677,E1 25.0825,E2 508.7472} C_DIS
LIN {X 60.1544,Y -104.4266,Z 131,A -63.9026,B 24.9597,C -1.4651,E1 25.0791,E2 510.1172} C_DIS
LIN {X 57.4422,Y -105.9428,Z 131,A -65.4608,B 24.9601,C -1.4586,E1 25.0753,E2 511.6862} C_DIS
LIN {X 53.8566,Y -107.8093,Z 131,A -67.3996,B 24.9604,C -1.4545,E1 25.0705,E2 513.6293} C_DIS
LIN {X 46.4979,Y -111.1818,Z 131,A -71.0368,B 24.9601,C -1.4586,E1 25.0613,E2 517.2478} C_DIS
LIN {X 43.4586,Y -112.4048,Z 131,A -73.6298,B 24.9629,C -1.4075,E1 25.0542,E2 519.956} C_DIS
LIN {X 37.7808,Y -114.438,Z 131,A -75.3795,B 24.9603,C -1.4565,E1 25.0499,E2 521.5864} C_DIS
LIN {X 34.9662,Y -115.3298,Z 131,A -77.0105,B 24.9609,C -1.444,E1 25.0455,E2 523.2439} C_DIS
LIN {X 31.2611,Y -116.3877,Z 131,A -79.0249,B 24.9615,C -1.4334,E1 25.04,E2 525.2802} C_DIS
LIN {X 26.2817,Y -117.613,Z 131,A -81.3406,B 24.9613,C -1.4368,E1 25.0337,E2 527.5847} C_DIS
LIN {X 20.1903,Y -118.8099,Z 131,A -84.1721,B 24.9612,C -1.44,E1 25.026,E2 530.4055} C_DIS
LIN {X 14.5573,Y -119.631,Z 131,A -86.9659,B 24.9615,C -1.434,E1 25.0182,E2 533.2108} C_DIS
LIN {X 6.0605,Y -120.3606,Z 131,A -91.8893,B 24.9637,C -1.3921,E1 25.0043,E2 538.2313} C_DIS
LIN {X 0.8351,Y -120.4889,Z 131,A -92.1351,B 24.9581,C -1.4959,E1 25.0043,E2 538.2313} C_DIS
Enddeposition()
LIN {X 0.8351,Y -120.4889,Z 131,A -92.1351,B 24.9581,C -1.4959,E1 25.0043,E2 538.2313} C_DIS
Startdeposition()
$VEL.CP = VEL_PRINT
LIN {X 2.318,Y -119.6505,Z 131,A -91.4699,B 24.9574,C -1.5079,E1 25.0063,E2 537.5377} C_DIS
LIN {X 6.4532,Y -119.4989,Z 131,A -90.0089,B 24.9587,C -1.4842,E1 25.0101,E2 536.1334} C_DIS
LIN {X 12.6185,Y -119.005,Z 131,A -86.9773,B 24.9585,C -1.489,E1 25.0186,E2 533.092} C_DIS
LIN {X 16.3228,Y -118.5548,Z 131,A -85.2112,B 24.9585,C -1.4892,E1 25.0234,E2 531.3269} C_DIS
LIN {X 21.6587,Y -117.6962,Z 131,A -82.5887,B 24.9582,C -1.4929,E1 25.0307,E2 528.6985} C_DIS
LIN {X 25.7398,Y -116.8712,Z 131,A -80.8185,B 24.9587,C -1.4841,E1 25.0355,E2 526.9513} C_DIS
LIN {X 28.7361,Y -116.1711,Z 131,A -79.2906,B 24.9585,C -1.4881,E1 25.0396,E2 525.416} C_DIS
LIN {X 32.0774,Y -115.2933,Z 131,A -77.4832,B 24.958,C -1.4972,E1 25.0445,E2 523.59} C_DIS
LIN {X 35.8895,Y -114.1647,Z 131,A -75.6982,B 24.9582,C -1.4938,E1 25.0493,E2 521.8163} C_DIS
LIN {X 38.2559,Y -113.3926,Z 131,A -74.2044,B 24.9573,C -1.5098,E1 25.0533,E2 520.2876} C_DIS
LIN {X 42.7918,Y -111.7603,Z 131,A -72.1548,B 24.9578,C -1.5005,E1 25.0586,E2 518.2643} C_DIS
LIN {X 46.0848,Y -110.4437,Z 131,A -70.4717,B 24.9578,C -1.5022,E1 25.063,E2 516.5809} C_DIS
LIN {X 49.1285,Y -109.1237,Z 131,A -68.588,B 24.9568,C -1.5189,E1 25.0679,E2 514.6624} C_DIS
LIN {X 52.0475,Y -107.7621,Z 131,A -67.274,B 24.9573,C -1.5104,E1 25.0711,E2 513.372} C_DIS
LIN {X 55.433,Y -106.0595,Z 131,A -65.668,B 24.9577,C -1.5035,E1 25.0751,E2 511.7868} C_DIS
LIN {X 57.3691,Y -105.0251,Z 131,A -64.0981,B 24.9561,C -1.5305,E1 25.0791,E2 510.1577} C_DIS
LIN {X 60.5971,Y -103.1969,Z 131,A -61.8582,B 24.9546,C -1.5565,E1 25.0846,E2 507.8631} C_DIS
LIN {X 65.5738,Y -100.108,Z 131,A -59.8942,B 24.9567,C -1.5209,E1 25.089,E2 505.9897} C_DIS
LIN {X 69.0567,Y -97.7388,Z 131,A -58.0467,B 24.9569,C -1.5168,E1 25.0932,E2 504.1582} C_DIS
LIN {X 70.8817,Y -96.4226,Z 131,A -56.9736,B 24.9568,C -1.5189,E1 25.0956,E2 503.084} C_DIS
LIN {X 74.1725,Y -93.9148,Z 131,A -54.8229,B 24.9561,C -1.5315,E1 25.1004,E2 500.9114} C_DIS
LIN {X 77.3636,Y -91.3036,Z 131,A -52.9172,B 24.956,C -1.5326,E1 25.1045,E2 499.0103} C_DIS
LIN {X 79.4987,Y -89.4512,Z 131,A -51.3804,B 24.9553,C -1.5447,E1 25.1077,E2 497.451} C_DIS
LIN {X 84.247,Y -84.9944,Z 131,A -48.42,B 24.9553,C -1.5446,E1 25.1137,E2 494.5032} C_DIS
LIN {X 87.0077,Y -82.1654,Z 131,A -46.0304,B 24.9536,C -1.5739,E1 25.1184,E2 492.0548} C_DIS
LIN {X 89.9787,Y -78.9007,Z 131,A -44.2275,B 24.9542,C -1.564,E1 25.1216,E2 490.2832} C_DIS
LIN {X 92.9734,Y -75.3493,Z 131,A -42.1984,B 24.9544,C -1.5603,E1 25.1252,E2 488.2723} C_DIS
LIN {X 95.3719,Y -72.2889,Z 131,A -40.2578,B 24.9539,C -1.5693,E1 25.1285,E2 486.3196} C_DIS
LIN {X 98.1351,Y -68.4909,Z 131,A -38.2574,B 24.9542,C -1.5634,E1 25.1317,E2 484.3431} C_DIS
LIN {X 100.2155,Y -65.4107,Z 131,A -36.5301,B 24.9541,C -1.5658,E1 25.1344,E2 482.6185} C_DIS
LIN {X 101.5358,Y -63.3403,Z 131,A -35.3908,B 24.954,C -1.5675,E1 25.1361,E2 481.4811} C_DIS
LIN {X 103.3478,Y -60.3385,Z 131,A -33.6934,B 24.9536,C -1.5733,E1 25.1385,E2 479.7786} C_DIS
LIN {X 105.6054,Y -56.2941,Z 131,A -31.4038,B 24.953,C -1.5835,E1 25.1416,E2 477.4771} C_DIS
LIN {X 107.2507,Y -53.093,Z 131,A -29.8042,B 24.953,C -1.5826,E1 25.1436,E2 475.8881} C_DIS
LIN {X 108.2852,Y -50.9497,Z 131,A -28.4753,B 24.9523,C -1.5954,E1 25.1453,E2 474.536} C_DIS
LIN {X 109.9567,Y -47.2346,Z 131,A -26.5427,B 24.952,C -1.6006,E1 25.1474,E2 472.6019} C_DIS
LIN {X 111.4837,Y -43.5067,Z 131,A -24.6407,B 24.9517,C -1.6053,E1 25.1494,E2 470.6993} C_DIS
LIN {X 112.89,Y -39.7163,Z 131,A -22.6964,B 24.9513,C -1.6118,E1 25.1512,E2 468.7505} C_DIS
LIN {X 114.2104,Y -35.7435,Z 131,A -20.7174,B 24.951,C -1.6169,E1 25.1529,E2 466.7706} C_DIS
LIN {X 115.2219,Y -32.3341,Z 131,A -19.0124,B 24.9507,C -1.6225,E1 25.1543,E2 465.0622} C_DIS
LIN {X 116.2832,Y -28.2811,Z 131,A -17.1753,B 24.9507,C -1.6206,E1 25.1555,E2 463.2403} C_DIS
LIN {X 117.0712,Y -24.8171,Z 131,A -15.4874,B 24.9505,C -1.6255,E1 25.1565,E2 461.5507} C_DIS
LIN {X 117.5538,Y -22.4172,Z 131,A -14.3618,B 24.9504,C -1.627,E1 25.1571,E2 460.428} C_DIS
LIN {X 117.9725,Y -20.0994,Z 131,A -13.2457,B 24.9502,C -1.6301,E1 25.1577,E2 459.3111} C_DIS
LIN {X 118.3222,Y -17.9252,Z 131,A -12.0165,B 24.9495,C -1.6422,E1 25.1582,E2 458.0606} C_DIS
LIN {X 118.8401,Y -14.0917,Z 131,A -10.251,B 24.9494,C -1.644,E1 25.1588,E2 456.3013} C_DIS
LIN {X 119.187,Y -10.7732,Z 131,A -8.4372,B 24.9484,C -1.66,E1 25.1593,E2 454.4605} C_DIS
LIN {X 119.5028,Y -6.3785,Z 131,A -6.57,B 24.9487,C -1.6549,E1 25.1596,E2 452.6166} C_DIS
LIN {X 119.6552,Y -2.0598,Z 131,A -4.479,B 24.9482,C -1.6628,E1 25.1598,E2 450.5194} C_DIS
LIN {X 119.6626,Y 1.5375,Z 131,A -2.8389,B 24.9481,C -1.6643,E1 25.1598,E2 448.8854} C_DIS
LIN {X 119.5794,Y 4.7166,Z 131,A -1.112,B 24.9471,C -1.6794,E1 25.1596,E2 447.1331} C_DIS
LIN {X 119.2731,Y 9.7715,Z 131,A 1.106,B 24.9473,C -1.6771,E1 25.1592,E2 444.9339} C_DIS
LIN {X 118.9474,Y 13.1612,Z 131,A 2.8982,B 24.9465,C -1.6904,E1 25.1586,E2 443.1209} C_DIS
LIN {X 118.2711,Y 18.2595,Z 131,A 5.3149,B 24.9461,C -1.696,E1 25.1577,E2 440.7051} C_DIS
LIN {X 117.6233,Y 22.0528,Z 131,A 7.0814,B 24.946,C -1.6981,E1 25.1568,E2 438.944} C_DIS
LIN {X 116.771,Y 26.1962,Z 131,A 9.1952,B 24.9453,C -1.7089,E1 25.1555,E2 436.8172} C_DIS
LIN {X 115.6823,Y 30.6457,Z 131,A 11.2247,B 24.9453,C -1.7076,E1 25.1542,E2 434.8023} C_DIS
LIN {X 114.8414,Y 33.6608,Z 131,A 12.7837,B 24.9449,C -1.7152,E1 25.1529,E2 433.2343} C_DIS
LIN {X 113.556,Y 37.7718,Z 131,A 14.8354,B 24.9445,C -1.721,E1 25.1512,E2 431.1806} C_DIS
LIN {X 112.1812,Y 41.6762,Z 131,A 16.9986,B 24.9435,C -1.7359,E1 25.1491,E2 428.9943} C_DIS
LIN {X 110.4809,Y 45.9963,Z 131,A 19.0034,B 24.9438,C -1.7317,E1 25.147,E2 427.0105} C_DIS
LIN {X 108.8479,Y 49.7357,Z 131,A 20.9365,B 24.9435,C -1.7364,E1 25.1448,E2 425.0769} C_DIS
LIN {X 107.5561,Y 52.4709,Z 131,A 22.2549,B 24.9436,C -1.7342,E1 25.1432,E2 423.7709} C_DIS
LIN {X 105.9608,Y 55.6218,Z 131,A 23.9493,B 24.9433,C -1.7391,E1 25.141,E2 422.0737} C_DIS
LIN {X 104.2049,Y 58.8472,Z 131,A 25.6375,B 24.9433,C -1.7405,E1 25.1388,E2 420.391} C_DIS
LIN {X 102.4182,Y 61.9032,Z 131,A 27.4455,B 24.9426,C -1.7507,E1 25.1362,E2 418.5684} C_DIS
LIN {X 100.32,Y 65.2492,Z 131,A 29.3696,B 24.9421,C -1.7573,E1 25.1333,E2 416.6384} C_DIS
LIN {X 98.0451,Y 68.6195,Z 131,A 31.3467,B 24.9417,C -1.7638,E1 25.1301,E2 414.6557} C_DIS
LIN {X 95.5229,Y 72.0892,Z 131,A 33.3618,B 24.9415,C -1.7671,E1 25.1268,E2 412.6425} C_DIS
LIN {X 93.1777,Y 75.097,Z 131,A 35.1463,B 24.9413,C -1.7695,E1 25.1237,E2 410.8607} C_DIS
LIN {X 90.8654,Y 77.879,Z 131,A 36.8703,B 24.9411,C -1.7732,E1 25.1206,E2 409.1358} C_DIS
LIN {X 88.3405,Y 80.7306,Z 131,A 38.645,B 24.9409,C -1.775,E1 25.1173,E2 407.3646} C_DIS
LIN {X 85.922,Y 83.3,Z 131,A 40.4621,B 24.9403,C -1.7849,E1 25.1137,E2 405.5319} C_DIS
LIN {X 83.294,Y 85.9278,Z 131,A 43.2092,B 24.9368,C -1.8358,E1 25.108,E2 402.6761} C_DIS
LIN {X 78.1604,Y 90.6226,Z 131,A 45.4728,B 24.9399,C -1.7907,E1 25.1035,E2 400.5281} C_DIS
LIN {X 75.237,Y 93.0644,Z 131,A 47.2565,B 24.9398,C -1.7922,E1 25.0996,E2 398.7475} C_DIS
LIN {X 72.0816,Y 95.5287,Z 131,A 49.1927,B 24.9395,C -1.7967,E1 25.0953,E2 396.8078} C_DIS
LIN {X 68.7543,Y 97.9506,Z 131,A 51.0947,B 24.9395,C -1.7969,E1 25.091,E2 394.9121} C_DIS
LIN {X 65.7299,Y 100.005,Z 131,A 52.8958,B 24.9391,C -1.8021,E1 25.0868,E2 393.1045} C_DIS
LIN {X 62.2883,Y 102.184,Z 131,A 54.8312,B 24.939,C -1.8045,E1 25.0822,E2 391.1697} C_DIS
LIN {X 59.7544,Y 103.687,Z 131,A 56.3195,B 24.9386,C -1.8102,E1 25.0786,E2 389.6723} C_DIS
LIN {X 55.8397,Y 105.8465,Z 131,A 58.3679,B 24.9386,C -1.8088,E1 25.0736,E2 387.6331} C_DIS
LIN {X 52.5547,Y 107.5151,Z 131,A 60.044,B 24.9388,C -1.8069,E1 25.0695,E2 385.966} C_DIS
LIN {X 49.3196,Y 109.0373,Z 131,A 61.8737,B 24.9383,C -1.8145,E1 25.0648,E2 384.123} C_DIS
LIN {X 45.5671,Y 110.6577,Z 131,A 63.7787,B 24.9383,C -1.8142,E1 25.0599,E2 382.2233} C_DIS
LIN {X 42.9702,Y 111.6925,Z 131,A 65.12,B 24.9383,C -1.8157,E1 25.0564,E2 380.8815} C_DIS
LIN {X 39.2837,Y 113.0409,Z 131,A 67.0256,B 24.938,C -1.8186,E1 25.0514,E2 378.9727} C_DIS
LIN {X 35.3995,Y 114.3169,Z 131,A 68.9862,B 24.9379,C -1.8203,E1 25.0462,E2 377.0116} C_DIS
LIN {X 31.9102,Y 115.3397,Z 131,A 70.7537,B 24.9377,C -1.8228,E1 25.0414,E2 375.2413} C_DIS
LIN {X 28.2163,Y 116.299,Z 131,A 72.5234,B 24.9378,C -1.8212,E1 25.0366,E2 373.478} C_DIS
LIN {X 25.0385,Y 117.0246,Z 131,A 73.9241,B 24.9383,C -1.8146,E1 25.0329,E2 372.0947} C_DIS
LIN {X 22.5357,Y 117.5312,Z 131,A 75.316,B 24.9377,C -1.823,E1 25.029,E2 370.6847} C_DIS
LIN {X 18.4084,Y 118.2483,Z 131,A 77.3481,B 24.9376,C -1.8249,E1 25.0234,E2 368.6502} C_DIS
LIN {X 14.1963,Y 118.8278,Z 131,A 79.1085,B 24.9384,C -1.8127,E1 25.0186,E2 366.9201} C_DIS
LIN {X 11.7483,Y 119.0946,Z 131,A 80.5676,B 24.9375,C -1.8257,E1 25.0145,E2 365.4311} C_DIS
LIN {X 7.6752,Y 119.4267,Z 131,A 82.4076,B 24.9379,C -1.8204,E1 25.0094,E2 363.6045} C_DIS
LIN {X 4.3459,Y 119.5942,Z 131,A 84.0061,B 24.9379,C -1.8204,E1 25.0049,E2 362.0064} C_DIS
LIN {X 0.2296,Y 119.6723,Z 131,A 86.1329,B 24.9374,C -1.8272,E1 24.9989,E2 359.8637} C_DIS
LIN {X -4.5374,Y 119.5868,Z 131,A 88.3641,B 24.9376,C -1.8242,E1 24.9927,E2 357.6393} C_DIS
LIN {X -9.0023,Y 119.3335,Z 131,A 90.4436,B 24.9379,C -1.8206,E1 24.9869,E2 355.5678} C_DIS
LIN {X -11.7939,Y 119.0902,Z 131,A 91.8685,B 24.9377,C -1.8237,E1 24.983,E2 354.1348} C_DIS
LIN {X -15.975,Y 118.6014,Z 131,A 93.8612,B 24.9378,C -1.8214,E1 24.9775,E2 352.1461} C_DIS
LIN {X -19.8954,Y 118.0075,Z 131,A 95.7153,B 24.938,C -1.8181,E1 24.9724,E2 350.2981} C_DIS
LIN {X -25.0978,Y 117.0117,Z 131,A 98.2007,B 24.9383,C -1.8137,E1 24.9656,E2 347.8204} C_DIS
LIN {X -27.832,Y 116.391,Z 131,A 99.6614,B 24.9381,C -1.8177,E1 24.9616,E2 346.3481} C_DIS
LIN {X -31.2743,Y 115.5138,Z 131,A 101.3603,B 24.9381,C -1.8159,E1 24.957,E2 344.651} C_DIS
LIN {X -35.259,Y 114.3602,Z 131,A 103.3425,B 24.9384,C -1.8135,E1 24.9517,E2 342.6713} C_DIS
LIN {X -39.959,Y 112.8048,Z 131,A 105.67,B 24.9387,C -1.8086,E1 24.9456,E2 340.3509} C_DIS
LIN {X -42.7762,Y 111.7663,Z 131,A 107.1705,B 24.9387,C -1.8095,E1 24.9416,E2 338.8451} C_DIS
LIN {X -45.9524,Y 110.4991,Z 131,A 108.6062,B 24.9394,C -1.7983,E1 24.938,E2 337.4329} C_DIS
LIN {X -48.1682,Y 109.5514,Z 131,A 109.9905,B 24.9388,C -1.8067,E1 24.9344,E2 336.0253} C_DIS
LIN {X -51.2595,Y 108.1389,Z 131,A 111.3794,B 24.9397,C -1.7937,E1 24.9309,E2 334.6639} C_DIS
LIN {X -53.7265,Y 106.9345,Z 131,A 112.9751,B 24.939,C -1.8039,E1 24.9269,E2 333.0396} C_DIS
LIN {X -57.6071,Y 104.8948,Z 131,A 116.0654,B 24.9362,C -1.8442,E1 24.9191,E2 329.8447} C_DIS
LIN {X -63.5873,Y 101.3817,Z 131,A 118.3554,B 24.9398,C -1.7923,E1 24.9139,E2 327.6709} C_DIS
LIN {X -67.029,Y 99.1394,Z 131,A 120.3484,B 24.94,C -1.7896,E1 24.9092,E2 325.6778} C_DIS
LIN {X -69.691,Y 97.286,Z 131,A 122.0875,B 24.9396,C -1.7945,E1 24.9053,E2 323.9209} C_DIS
LIN {X -72.5215,Y 95.1959,Z 131,A 124.2974,B 24.9383,C -1.8139,E1 24.9003,E2 321.6569} C_DIS
LIN {X -76.7117,Y 91.8518,Z 131,A 126.1659,B 24.9408,C -1.7776,E1 24.8964,E2 319.8676} C_DIS
LIN {X -79.7296,Y 89.2444,Z 131,A 127.8417,B 24.9417,C -1.7632,E1 24.8929,E2 318.2197} C_DIS
LIN {X -81.3963,Y 87.7277,Z 131,A 129.1156,B 24.9413,C -1.769,E1 24.8903,E2 316.9267} C_DIS
LIN {X -84.0099,Y 85.2283,Z 131,A 130.84,B 24.9416,C -1.7645,E1 24.8868,E2 315.2058} C_DIS
LIN {X -86.4929,Y 82.7077,Z 131,A 132.5354,B 24.9419,C -1.7604,E1 24.8835,E2 313.513} C_DIS
LIN {X -89.0952,Y 79.8962,Z 131,A 134.3647,B 24.9422,C -1.7555,E1 24.8801,E2 311.6872} C_DIS
LIN {X -90.8898,Y 77.8502,Z 131,A 136.1888,B 24.941,C -1.7745,E1 24.8767,E2 309.8094} C_DIS
LIN {X -93.4623,Y 74.7416,Z 131,A 137.695,B 24.9425,C -1.751,E1 24.8741,E2 308.3522} C_DIS
LIN {X -95.7005,Y 71.854,Z 131,A 139.5421,B 24.9425,C -1.7505,E1 24.871,E2 306.4976} C_DIS
LIN {X -98.3624,Y 68.1648,Z 131,A 141.3746,B 24.9439,C -1.7296,E1 24.8681,E2 304.7059} C_DIS
LIN {X -100.2316,Y 65.3858,Z 131,A 143.1618,B 24.9437,C -1.7329,E1 24.8653,E2 302.9018} C_DIS
LIN {X -102.0736,Y 62.4697,Z 131,A 144.8007,B 24.9441,C -1.7276,E1 24.8629,E2 301.2671} C_DIS
LIN {X -103.4766,Y 60.1178,Z 131,A 146.533,B 24.9431,C -1.7418,E1 24.8604,E2 299.4921} C_DIS
LIN {X -105.146,Y 57.148,Z 131,A 147.8962,B 24.9442,C -1.7255,E1 24.8586,E2 298.1606} C_DIS
LIN {X -106.8013,Y 53.9924,Z 131,A 149.6246,B 24.9445,C -1.7213,E1 24.8564,E2 296.4329} C_DIS
LIN {X -108.3119,Y 50.8925,Z 131,A 151.8104,B 24.9433,C -1.7392,E1 24.8538,E2 294.1926} C_DIS
LIN {X -110.1716,Y 46.7295,Z 131,A 153.4341,B 24.9453,C -1.7085,E1 24.852,E2 292.633} C_DIS
LIN {X -111.6668,Y 43.0375,Z 131,A 155.4184,B 24.9455,C -1.7059,E1 24.85,E2 290.644} C_DIS
LIN {X -112.9172,Y 39.6387,Z 131,A 156.9023,B 24.9465,C -1.6898,E1 24.8486,E2 289.1899} C_DIS
LIN {X -114.1818,Y 35.8358,Z 131,A 159.0229,B 24.9463,C -1.6923,E1 24.8468,E2 287.0513} C_DIS
LIN {X -115.3706,Y 31.799,Z 131,A 161.8288,B 24.9446,C -1.7196,E1 24.8446,E2 284.1639} C_DIS
LIN {X -116.7003,Y 26.5051,Z 131,A 163.7392,B 24.947,C -1.6811,E1 24.8435,E2 282.3341} C_DIS
LIN {X -117.5881,Y 22.2374,Z 131,A 165.8233,B 24.9475,C -1.6742,E1 24.8423,E2 280.2542} C_DIS
LIN {X -118.2816,Y 18.1911,Z 131,A 167.6686,B 24.9482,C -1.6627,E1 24.8415,E2 278.4253} C_DIS
LIN {X -118.7887,Y 14.5193,Z 131,A 169.5828,B 24.9482,C -1.6628,E1 24.8408,E2 276.4995} C_DIS
LIN {X -119.1734,Y 10.923,Z 131,A 171.3362,B 24.9485,C -1.6581,E1 24.8403,E2 274.7469} C_DIS
LIN {X -119.49,Y 6.6125,Z 131,A 173.3229,B 24.9491,C -1.6478,E1 24.84,E2 272.7727} C_DIS
LIN {X -119.6344,Y 3.0314,Z 131,A 175.0627,B 24.9494,C -1.6432,E1 24.8398,E2 271.0334} C_DIS
LIN {X -119.6704,Y -0.6404,Z 131,A 176.8589,B 24.9497,C -1.6391,E1 24.8398,E2 269.2361} C_DIS
LIN {X -119.5934,Y -4.3716,Z 131,A 178.7441,B 24.9497,C -1.6374,E1 24.84,E2 267.3436} C_DIS
LIN {X -119.4175,Y -7.8102,Z 131,A -179.6244,B 24.9501,C -1.6313,E1 24.8402,E2 265.7167} C_DIS
LIN {X -119.0627,Y -12.0709,Z 131,A -177.5905,B 24.9506,C -1.6242,E1 24.8408,E2 263.6878} C_DIS
LIN {X -118.6021,Y -15.9696,Z 131,A -175.6451,B 24.9508,C -1.6209,E1 24.8414,E2 261.7384} C_DIS
LIN {X -117.98,Y -20.0562,Z 131,A -173.7334,B 24.9513,C -1.6117,E1 24.8423,E2 259.8373} C_DIS
LIN {X -117.2274,Y -24.0692,Z 131,A -171.7161,B 24.9515,C -1.6082,E1 24.8434,E2 257.8164} C_DIS
LIN {X -116.3133,Y -28.1577,Z 131,A -169.7926,B 24.9521,C -1.5984,E1 24.8446,E2 255.905} C_DIS
LIN {X -115.7232,Y -30.493,Z 131,A -168.0643,B 24.9509,C -1.6195,E1 24.8459,E2 254.1164} C_DIS
LIN {X -114.5875,Y -34.5144,Z 131,A -166.5763,B 24.9526,C -1.5913,E1 24.847,E2 252.687} C_DIS
LIN {X -113.4421,Y -38.1096,Z 131,A -164.7688,B 24.9529,C -1.5858,E1 24.8486,E2 250.8822} C_DIS
LIN {X -110.9034,Y -44.9672,Z 131,A -161.3554,B 24.9537,C -1.5716,E1 24.8519,E2 247.4836} C_DIS
LIN {X -109.6583,Y -47.9229,Z 131,A -159.7081,B 24.9537,C -1.5719,E1 24.8537,E2 245.8264} C_DIS
LIN {X -108.09,Y -51.362,Z 131,A -157.7957,B 24.9537,C -1.5711,E1 24.856,E2 243.9053} C_DIS
LIN {X -106.418,Y -54.7417,Z 131,A -155.984,B 24.954,C -1.5663,E1 24.8583,E2 242.0954} C_DIS
LIN {X -104.8313,Y -57.7233,Z 131,A -154.3277,B 24.9542,C -1.5635,E1 24.8605,E2 240.437} C_DIS
LIN {X -103.064,Y -60.8227,Z 131,A -152.71,B 24.9547,C -1.555,E1 24.8628,E2 238.8313} C_DIS
LIN {X -101.1792,Y -63.9086,Z 131,A -151.0829,B 24.9552,C -1.5459,E1 24.8651,E2 237.2175} C_DIS
LIN {X -99.2925,Y -66.8015,Z 131,A -148.9303,B 24.9542,C -1.5633,E1 24.8685,E2 235.0128} C_DIS
LIN {X -97.3025,Y -69.668,Z 131,A -146.4663,B 24.9524,C -1.5941,E1 24.8727,E2 232.4634} C_DIS
LIN {X -92.9702,Y -75.3533,Z 131,A -144.1344,B 24.9557,C -1.5376,E1 24.8766,E2 230.255} C_DIS
LIN {X -90.3031,Y -78.5301,Z 131,A -142.1486,B 24.956,C -1.533,E1 24.8802,E2 228.2712} C_DIS
LIN {X -87.0156,Y -82.157,Z 131,A -139.7683,B 24.9562,C -1.5293,E1 24.8847,E2 225.8892} C_DIS
LIN {X -84.1307,Y -85.1093,Z 131,A -138.073,B 24.9571,C -1.5127,E1 24.8879,E2 224.2262} C_DIS
LIN {X -81.442,Y -87.6852,Z 131,A -135.9674,B 24.9565,C -1.5232,E1 24.8923,E2 222.087} C_DIS
LIN {X -78.3405,Y -90.4671,Z 131,A -134.0665,B 24.957,C -1.5151,E1 24.8962,E2 220.1979} C_DIS
LIN {X -75.5757,Y -92.7889,Z 131,A -132.2547,B 24.957,C -1.5154,E1 24.9002,E2 218.3784} C_DIS
LIN {X -72.6581,Y -95.0916,Z 131,A -130.4695,B 24.9571,C -1.5124,E1 24.9041,E2 216.5937} C_DIS
LIN {X -69.242,Y -97.6066,Z 131,A -128.6393,B 24.9578,C -1.5,E1 24.9082,E2 214.7866} C_DIS
LIN {X -67.3036,Y -98.9537,Z 131,A -127.2821,B 24.9574,C -1.5082,E1 24.9114,E2 213.4054} C_DIS
LIN {X -63.7538,Y -101.2773,Z 131,A -125.3501,B 24.9578,C -1.5006,E1 24.9159,E2 211.4853} C_DIS
LIN {X -60.5547,Y -103.2216,Z 131,A -123.4495,B 24.9577,C -1.5028,E1 24.9205,E2 209.5737} C_DIS
LIN {X -57.0102,Y -105.2208,Z 131,A -121.5092,B 24.9579,C -1.4997,E1 24.9252,E2 207.6351} C_DIS
LIN {X -53.8416,Y -106.8769,Z 131,A -119.7956,B 24.9579,C -1.4976,E1 24.9295,E2 205.9219} C_DIS
LIN {X -50.1566,Y -108.6549,Z 131,A -117.8148,B 24.9581,C -1.4963,E1 24.9345,E2 203.9392} C_DIS
LIN {X -46.3122,Y -110.3478,Z 131,A -116.0623,B 24.9588,C -1.4824,E1 24.9389,E2 202.2156} C_DIS
LIN {X -43.5113,Y -111.4819,Z 131,A -114.3297,B 24.9582,C -1.4939,E1 24.9435,E2 200.4519} C_DIS
LIN {X -39.4237,Y -112.9921,Z 131,A -112.427,B 24.9588,C -1.4837,E1 24.9484,E2 198.5696} C_DIS
LIN {X -36.9521,Y -113.8251,Z 131,A -111.2138,B 24.9589,C -1.4811,E1 24.9516,E2 197.3604} C_DIS
LIN {X -33.824,Y -114.793,Z 131,A -109.466,B 24.9585,C -1.4881,E1 24.9563,E2 195.5929} C_DIS
LIN {X -30.3301,Y -115.7656,Z 131,A -107.8981,B 24.959,C -1.4793,E1 24.9605,E2 194.0434} C_DIS
LIN {X -27.9412,Y -116.365,Z 131,A -106.7205,B 24.959,C -1.4786,E1 24.9637,E2 192.8659} C_DIS
LIN {X -25.299,Y -116.9678,Z 131,A -105.2483,B 24.9586,C -1.486,E1 24.9678,E2 191.3743} C_DIS
LIN {X -21.3925,Y -117.7445,Z 131,A -103.3332,B 24.9586,C -1.4857,E1 24.973,E2 189.458} C_DIS
LIN {X -17.4733,Y -118.3906,Z 131,A -101.6411,B 24.9592,C -1.4754,E1 24.9776,E2 187.7886} C_DIS
LIN {X -15.0723,Y -118.7197,Z 131,A -100.1086,B 24.9583,C -1.4924,E1 24.982,E2 186.2147} C_DIS
LIN {X -10.5205,Y -119.2091,Z 131,A -98.132,B 24.9588,C -1.4823,E1 24.9874,E2 184.2611} C_DIS
LIN {X -6.6227,Y -119.4895,Z 131,A -96.1338,B 24.9585,C -1.4882,E1 24.993,E2 182.2482} C_DIS
LIN {X -0.4873,Y -119.6712,Z 131,A -93.3771,B 24.959,C -1.4802,E1 25.0007,E2 179.5102} C_DIS
LIN {X -0.4873,Y -119.6712,Z 131,A -93.3771,B 24.959,C -1.4802,E1 25.0007,E2 179.5102} C_DIS
Enddeposition()
LIN {X 0.8316,Y -118.8261,Z 131,A -93.3596,B 24.9597,C -1.4667,E1 25.0007,E2 179.5246} C_DIS
Startdeposition()
$VEL.CP = VEL_PRINT
LIN {X -2.9704,Y -118.7949,Z 131,A -95.2293,B 24.9598,C -1.4647,E1 24.9954,E2 181.3992} C_DIS
LIN {X -5.8621,Y -118.6872,Z 131,A -96.6516,B 24.9598,C -1.4633,E1 24.9914,E2 182.8251} C_DIS
LIN {X -8.8463,Y -118.5025,Z 131,A -98.1591,B 24.9601,C -1.4603,E1 24.9872,E2 184.3403} C_DIS
LIN {X -12.6268,Y -118.1587,Z 131,A -100.0376,B 24.9601,C -1.4583,E1 24.982,E2 186.2245} C_DIS
LIN {X -16.014,Y -117.748,Z 131,A -101.5732,B 24.9599,C -1.4636,E1 24.9777,E2 187.7488} C_DIS
LIN {X -18.977,Y -117.3067,Z 131,A -102.993,B 24.9598,C -1.4651,E1 24.9738,E2 189.1663} C_DIS
LIN {X -21.7559,Y -116.8241,Z 131,A -104.4004,B 24.9598,C -1.4634,E1 24.9699,E2 190.5792} C_DIS
LIN {X -24.694,Y -116.2381,Z 131,A -105.783,B 24.9597,C -1.4668,E1 24.9662,E2 191.9552} C_DIS
LIN {X -27.5459,Y -115.5951,Z 131,A -107.3016,B 24.9599,C -1.4627,E1 24.962,E2 193.4856} C_DIS
LIN {X -31.2752,Y -114.6428,Z 131,A -109.2002,B 24.9599,C -1.4619,E1 24.9569,E2 195.389} C_DIS
LIN {X -34.4971,Y -113.7151,Z 131,A -110.7263,B 24.9597,C -1.467,E1 24.9528,E2 196.9053} C_DIS
LIN {X -37.3561,Y -112.8079,Z 131,A -112.1526,B 24.9596,C -1.4691,E1 24.949,E2 198.3295} C_DIS
LIN {X -40.6885,Y -111.6492,Z 131,A -113.8512,B 24.9595,C -1.4707,E1 24.9446,E2 200.0276} C_DIS
LIN {X -43.1948,Y -110.703,Z 131,A -115.0419,B 24.9592,C -1.4764,E1 24.9415,E2 201.2072} C_DIS
LIN {X -45.4888,Y -109.7809,Z 131,A -116.3327,B 24.9593,C -1.4732,E1 24.9381,E2 202.5083} C_DIS
LIN {X -48.2423,Y -108.5987,Z 131,A -117.7778,B 24.9593,C -1.4748,E1 24.9344,E2 203.9531} C_DIS
LIN {X -51.1066,Y -107.2804,Z 131,A -119.2361,B 24.959,C -1.4793,E1 24.9308,E2 205.4044} C_DIS
LIN {X -53.4212,Y -106.1472,Z 131,A -120.555,B 24.9591,C -1.4775,E1 24.9274,E2 206.7311} C_DIS
LIN {X -56.095,Y -104.7585,Z 131,A -122.1687,B 24.9594,C -1.4724,E1 24.9234,E2 208.3614} C_DIS
LIN {X -59.3984,Y -102.922,Z 131,A -123.9642,B 24.9592,C -1.4761,E1 24.9191,E2 210.1533} C_DIS
LIN {X -62.4217,Y -101.1167,Z 131,A -125.5594,B 24.9588,C -1.4831,E1 24.9153,E2 211.7368} C_DIS
LIN {X -65.4311,Y -99.195,Z 131,A -127.3992,B 24.9589,C -1.4808,E1 24.9109,E2 213.5882} C_DIS
LIN {X -68.4194,Y -97.159,Z 131,A -129.0488,B 24.9585,C -1.4877,E1 24.9072,E2 215.2267} C_DIS
LIN {X -70.8478,Y -95.4023,Z 131,A -130.635,B 24.9587,C -1.4842,E1 24.9036,E2 216.8271} C_DIS
LIN {X -73.7265,Y -93.1959,Z 131,A -132.388,B 24.9586,C -1.4872,E1 24.8997,E2 218.5794} C_DIS
LIN {X -77.1011,Y -90.4239,Z 131,A -134.4966,B 24.9583,C -1.4911,E1 24.8952,E2 220.6866} C_DIS
LIN {X -80.2248,Y -87.664,Z 131,A -136.3984,B 24.9579,C -1.4998,E1 24.8913,E2 222.5754} C_DIS
LIN {X -83.0001,Y -85.0416,Z 131,A -138.3874,B 24.9579,C -1.4973,E1 24.8872,E2 224.5785} C_DIS
LIN {X -86.0921,Y -81.9098,Z 131,A -140.5018,B 24.9577,C -1.5023,E1 24.8831,E2 226.6902} C_DIS
LIN {X -89.0247,Y -78.7127,Z 131,A -142.6127,B 24.9575,C -1.5062,E1 24.8792,E2 228.8011} C_DIS
LIN {X -91.8871,Y -75.3513,Z 131,A -144.7459,B 24.9572,C -1.5111,E1 24.8754,E2 230.9326} C_DIS
LIN {X -94.1784,Y -72.466,Z 131,A -146.5106,B 24.9569,C -1.5159,E1 24.8723,E2 232.694} C_DIS
LIN {X -96.0535,Y -69.9621,Z 131,A -148.0001,B 24.9567,C -1.5205,E1 24.8699,E2 234.1799} C_DIS
LIN {X -98.0426,Y -67.1466,Z 131,A -149.5274,B 24.9561,C -1.5305,E1 24.8675,E2 235.691} C_DIS
LIN {X -99.6103,Y -64.7985,Z 131,A -150.9438,B 24.9561,C -1.5317,E1 24.8653,E2 237.1117} C_DIS
LIN {X -101.2146,Y -62.264,Z 131,A -152.3911,B 24.9558,C -1.5354,E1 24.8631,E2 238.5573} C_DIS
LIN {X -102.709,Y -59.7651,Z 131,A -153.7714,B 24.9556,C -1.5403,E1 24.8612,E2 239.9333} C_DIS
LIN {X -104.1003,Y -57.3079,Z 131,A -155.1963,B 24.9555,C -1.5413,E1 24.8592,E2 241.3632} C_DIS
LIN {X -105.7809,Y -54.1414,Z 131,A -156.757,B 24.9548,C -1.5532,E1 24.8573,E2 242.9037} C_DIS
LIN {X -106.8346,Y -52.0326,Z 131,A -158.0271,B 24.9549,C -1.5508,E1 24.8557,E2 244.1865} C_DIS
LIN {X -108.0408,Y -49.4798,Z 131,A -159.4758,B 24.9549,C -1.551,E1 24.8539,E2 245.6426} C_DIS
LIN {X -109.256,Y -46.7367,Z 131,A -160.925,B 24.9547,C -1.5551,E1 24.8523,E2 247.09} C_DIS
LIN {X -110.3858,Y -44.0004,Z 131,A -162.2702,B 24.9542,C -1.5628,E1 24.8509,E2 248.4245} C_DIS
LIN {X -111.4248,Y -41.298,Z 131,A -163.6973,B 24.9541,C -1.5656,E1 24.8495,E2 249.8528} C_DIS
LIN {X -112.5544,Y -38.1106,Z 131,A -165.4133,B 24.954,C -1.567,E1 24.8479,E2 251.5753} C_DIS
LIN {X -113.7114,Y -34.5092,Z 131,A -167.2337,B 24.9537,C -1.5727,E1 24.8464,E2 253.3926} C_DIS
LIN {X -114.6802,Y -31.1368,Z 131,A -168.7413,B 24.9529,C -1.5856,E1 24.8453,E2 254.8782} C_DIS
LIN {X -115.2702,Y -28.876,Z 131,A -170.2015,B 24.9535,C -1.5752,E1 24.8443,E2 256.3717} C_DIS
LIN {X -116.1316,Y -25.1878,Z 131,A -172.0152,B 24.9531,C -1.5815,E1 24.8432,E2 258.1811} C_DIS
LIN {X -116.8254,Y -21.7491,Z 131,A -173.6627,B 24.9527,C -1.5886,E1 24.8423,E2 259.8213} C_DIS
LIN {X -117.3229,Y -18.8774,Z 131,A -174.9881,B 24.9522,C -1.5964,E1 24.8417,E2 261.136} C_DIS
LIN {X -117.8533,Y -15.2213,Z 131,A -176.9232,B 24.9522,C -1.5958,E1 24.8409,E2 263.0842} C_DIS
LIN {X -118.2711,Y -11.5299,Z 131,A -178.5588,B 24.9516,C -1.608,E1 24.8405,E2 264.7004} C_DIS
LIN {X -118.5107,Y -8.741,Z 131,A -179.992,B 24.9515,C -1.6089,E1 24.8401,E2 266.1402} C_DIS
LIN {X -118.7154,Y -5.2612,Z 131,A 178.5304,B 24.9507,C -1.6228,E1 24.8399,E2 267.5934} C_DIS
LIN {X -118.7963,Y -2.9099,Z 131,A 177.1886,B 24.951,C -1.6179,E1 24.8399,E2 268.9551} C_DIS
LIN {X -118.8323,Y 0.099,Z 131,A 175.7417,B 24.9507,C -1.6228,E1 24.8398,E2 270.399} C_DIS
LIN {X -118.7941,Y 3.0044,Z 131,A 174.3898,B 24.9503,C -1.6294,E1 24.8398,E2 271.7432} C_DIS
LIN {X -118.6891,Y 5.8245,Z 131,A 172.8721,B 24.9503,C -1.6273,E1 24.84,E2 273.2749} C_DIS
LIN {X -118.4512,Y 9.5018,Z 131,A 171.0379,B 24.9502,C -1.6308,E1 24.8404,E2 275.112} C_DIS
LIN {X -118.1082,Y 13.102,Z 131,A 169.3831,B 24.9496,C -1.6401,E1 24.8409,E2 276.7543} C_DIS
LIN {X -117.726,Y 16.1782,Z 131,A 167.9432,B 24.9492,C -1.6473,E1 24.8414,E2 278.1859} C_DIS
LIN {X -117.31,Y 18.9566,Z 131,A 166.4568,B 24.9492,C -1.6463,E1 24.8421,E2 279.6836} C_DIS
LIN {X -116.7461,Y 22.165,Z 131,A 164.8591,B 24.949,C -1.6503,E1 24.8429,E2 281.2811} C_DIS
LIN {X -115.931,Y 26.0983,Z 131,A 162.9948,B 24.9484,C -1.6595,E1 24.8439,E2 283.1344} C_DIS
LIN {X -115.2403,Y 28.9963,Z 131,A 161.4681,B 24.9484,C -1.6604,E1 24.845,E2 284.6679} C_DIS
LIN {X -114.523,Y 31.7094,Z 131,A 160.216,B 24.9478,C -1.6689,E1 24.8459,E2 285.9069} C_DIS
LIN {X -113.6821,Y 34.6043,Z 131,A 158.7727,B 24.9475,C -1.674,E1 24.847,E2 287.3465} C_DIS
LIN {X -112.8031,Y 37.3708,Z 131,A 157.3435,B 24.9473,C -1.6772,E1 24.8483,E2 288.7763} C_DIS
LIN {X -111.8833,Y 40.0391,Z 131,A 155.9728,B 24.947,C -1.6811,E1 24.8495,E2 290.1455} C_DIS
LIN {X -110.8692,Y 42.7689,Z 131,A 154.3868,B 24.9472,C -1.6779,E1 24.8511,E2 291.7479} C_DIS
LIN {X -109.204,Y 46.8573,Z 131,A 152.3869,B 24.9465,C -1.6898,E1 24.8532,E2 293.7306} C_DIS
LIN {X -108.0287,Y 49.5062,Z 131,A 151.0247,B 24.9461,C -1.6956,E1 24.8548,E2 295.0866} C_DIS
LIN {X -106.7874,Y 52.1292,Z 131,A 149.6164,B 24.9459,C -1.6994,E1 24.8565,E2 296.4933} C_DIS
LIN {X -105.4824,Y 54.723,Z 131,A 148.1582,B 24.9458,C -1.7012,E1 24.8583,E2 297.9551} C_DIS
LIN {X -104.1137,Y 57.2834,Z 131,A 146.7074,B 24.9456,C -1.7032,E1 24.8603,E2 299.4087} C_DIS
LIN {X -102.6236,Y 59.9116,Z 131,A 145.3527,B 24.9451,C -1.7118,E1 24.8622,E2 300.7501} C_DIS
LIN {X -100.9536,Y 62.6844,Z 131,A 143.6425,B 24.9451,C -1.7101,E1 24.8647,E2 302.4732} C_DIS
LIN {X -98.7948,Y 66.0355,Z 131,A 141.8029,B 24.9446,C -1.7189,E1 24.8675,E2 304.3008} C_DIS
LIN {X -97.1528,Y 68.4281,Z 131,A 140.3891,B 24.9444,C -1.7222,E1 24.8697,E2 305.7137} C_DIS
LIN {X -95.3903,Y 70.8639,Z 131,A 138.7986,B 24.9445,C -1.7204,E1 24.8724,E2 307.3164} C_DIS
LIN {X -93.1129,Y 73.8315,Z 131,A 137.0878,B 24.944,C -1.7291,E1 24.8753,E2 309.0145} C_DIS
LIN {X -90.8215,Y 76.6321,Z 131,A 135.2495,B 24.944,C -1.7298,E1 24.8786,E2 310.8596} C_DIS
LIN {X -88.0137,Y 79.8415,Z 131,A 133.1665,B 24.9437,C -1.734,E1 24.8824,E2 312.9421} C_DIS
LIN {X -85.0519,Y 82.9896,Z 131,A 131.0479,B 24.9434,C -1.7377,E1 24.8865,E2 315.0609} C_DIS
LIN {X -81.9138,Y 86.0883,Z 131,A 128.928,B 24.9431,C -1.7431,E1 24.8908,E2 317.1768} C_DIS
LIN {X -78.7122,Y 89.0252,Z 131,A 126.8156,B 24.9428,C -1.7473,E1 24.8951,E2 319.2877} C_DIS
LIN {X -75.3188,Y 91.9136,Z 131,A 124.6735,B 24.9424,C -1.7524,E1 24.8997,E2 321.4259} C_DIS
LIN {X -71.9508,Y 94.5736,Z 131,A 122.7289,B 24.9418,C -1.7621,E1 24.904,E2 323.3544} C_DIS
LIN {X -69.5358,Y 96.3638,Z 131,A 121.2566,B 24.9417,C -1.7642,E1 24.9073,E2 324.827} C_DIS
LIN {X -67.1529,Y 98.0383,Z 131,A 119.8933,B 24.9414,C -1.7688,E1 24.9104,E2 326.184} C_DIS
LIN {X -64.2698,Y 99.9523,Z 131,A 118.2119,B 24.9412,C -1.7715,E1 24.9143,E2 327.8645} C_DIS
LIN {X -62.0358,Y 101.3536,Z 131,A 116.9666,B 24.9409,C -1.775,E1 24.9173,E2 329.1053} C_DIS
LIN {X -59.6751,Y 102.7616,Z 131,A 115.6123,B 24.9409,C -1.7762,E1 24.9205,E2 330.4609} C_DIS
LIN {X -57.2783,Y 104.1165,Z 131,A 114.2005,B 24.9409,C -1.7749,E1 24.924,E2 331.8798} C_DIS
LIN {X -54.63,Y 105.5308,Z 131,A 112.7783,B 24.9407,C -1.7785,E1 24.9275,E2 333.2975} C_DIS
LIN {X -52.031,Y 106.8354,Z 131,A 111.422,B 24.9404,C -1.7827,E1 24.9309,E2 334.6472} C_DIS
LIN {X -49.4792,Y 108.041,Z 131,A 110.0088,B 24.9404,C -1.7826,E1 24.9345,E2 336.0643} C_DIS
LIN {X -46.7126,Y 109.2662,Z 131,A 108.5506,B 24.9403,C -1.7848,E1 24.9382,E2 337.5207} C_DIS
LIN {X -44.0468,Y 110.3672,Z 131,A 107.2121,B 24.94,C -1.789,E1 24.9416,E2 338.8521} C_DIS
LIN {X -41.3304,Y 111.4128,Z 131,A 105.7832,B 24.94,C -1.7898,E1 24.9454,E2 340.2823} C_DIS
LIN {X -38.6732,Y 112.3634,Z 131,A 104.2326,B 24.9404,C -1.7833,E1 24.9495,E2 341.8513} C_DIS
LIN {X -35.5406,Y 113.3933,Z 131,A 102.8873,B 24.9396,C -1.7957,E1 24.953,E2 343.1693} C_DIS
LIN {X -33.002,Y 114.1572,Z 131,A 101.5314,B 24.9396,C -1.7938,E1 24.9567,E2 344.5321} C_DIS
LIN {X -30.2805,Y 114.9099,Z 131,A 100.1404,B 24.9396,C -1.7939,E1 24.9604,E2 345.925} C_DIS
LIN {X -27.3687,Y 115.6373,Z 131,A 98.6,B 24.9399,C -1.7912,E1 24.9646,E2 347.4739} C_DIS
LIN {X -24.4958,Y 116.2796,Z 131,A 97.2987,B 24.9394,C -1.7977,E1 24.9681,E2 348.7615} C_DIS
LIN {X -21.7313,Y 116.8288,Z 131,A 95.9021,B 24.9394,C -1.7971,E1 24.972,E2 350.161} C_DIS
LIN {X -18.8682,Y 117.3244,Z 131,A 94.5245,B 24.9394,C -1.7992,E1 24.9758,E2 351.535} C_DIS
LIN {X -15.9913,Y 117.7511,Z 131,A 93.0972,B 24.9394,C -1.799,E1 24.9797,E2 352.9639} C_DIS
LIN {X -12.9968,Y 118.1195,Z 131,A 91.6665,B 24.9392,C -1.8009,E1 24.9837,E2 354.3911} C_DIS
LIN {X -9.982,Y 118.4124,Z 131,A 90.2571,B 24.939,C -1.8038,E1 24.9876,E2 355.7941} C_DIS
LIN {X -7.1844,Y 118.6144,Z 131,A 88.7955,B 24.9393,C -1.7996,E1 24.9917,E2 357.2663} C_DIS
LIN {X -4.3683,Y 118.7524,Z 131,A 87.4591,B 24.9393,C -1.801,E1 24.9954,E2 358.5996} C_DIS
LIN {X -1.3248,Y 118.8248,Z 131,A 86.0546,B 24.939,C -1.8042,E1 24.9993,E2 359.9966} C_DIS
LIN {X 1.5741,Y 118.8214,Z 131,A 84.634,B 24.939,C -1.8034,E1 25.0033,E2 361.4189} C_DIS
LIN {X 4.3907,Y 118.7515,Z 131,A 83.2363,B 24.9391,C -1.8018,E1 25.0072,E2 362.8202} C_DIS
LIN {X 7.3803,Y 118.6027,Z 131,A 81.8267,B 24.9391,C -1.8033,E1 25.0111,E2 364.2256} C_DIS
LIN {X 10.3114,Y 118.3836,Z 131,A 80.429,B 24.939,C -1.8041,E1 25.015,E2 365.6208} C_DIS
LIN {X 13.1176,Y 118.1063,Z 131,A 78.9978,B 24.9392,C -1.8007,E1 25.019,E2 367.0591} C_DIS
LIN {X 16.003,Y 117.7495,Z 131,A 77.4982,B 24.9395,C -1.796,E1 25.0232,E2 368.5686} C_DIS
LIN {X 20.0967,Y 117.1201,Z 131,A 75.6239,B 24.9392,C -1.8009,E1 25.0283,E2 370.4295} C_DIS
LIN {X 23.188,Y 116.5475,Z 131,A 74.1227,B 24.9392,C -1.8009,E1 25.0324,E2 371.9289} C_DIS
LIN {X 26.2479,Y 115.8968,Z 131,A 72.4784,B 24.9397,C -1.794,E1 25.0369,E2 373.5874} C_DIS
LIN {X 30.2914,Y 114.9069,Z 131,A 70.5956,B 24.9394,C -1.7984,E1 25.042,E2 375.457} C_DIS
LIN {X 33.1819,Y 114.1055,Z 131,A 69.2064,B 24.9393,C -1.8,E1 25.0457,E2 376.8401} C_DIS
LIN {X 35.8852,Y 113.284,Z 131,A 67.6853,B 24.9398,C -1.7917,E1 25.0498,E2 378.3781} C_DIS
LIN {X 38.9902,Y 112.2529,Z 131,A 66.2085,B 24.9396,C -1.7949,E1 25.0537,E2 379.8444} C_DIS
LIN {X 41.5073,Y 111.3475,Z 131,A 64.9768,B 24.9396,C -1.7963,E1 25.0569,E2 381.0701} C_DIS
LIN {X 44.1347,Y 110.3319,Z 131,A 63.6071,B 24.9396,C -1.7944,E1 25.0605,E2 382.4412} C_DIS
LIN {X 46.8265,Y 109.2173,Z 131,A 62.1586,B 24.9399,C -1.7909,E1 25.0642,E2 383.8948} C_DIS
LIN {X 49.4806,Y 108.0404,Z 131,A 60.694,B 24.9402,C -1.7863,E1 25.0679,E2 385.3665} C_DIS
LIN {X 52.1227,Y 106.7906,Z 131,A 59.2539,B 24.9404,C -1.7831,E1 25.0716,E2 386.8104} C_DIS
LIN {X 55.6143,Y 105.0151,Z 131,A 57.4024,B 24.9404,C -1.7823,E1 25.0762,E2 388.6587} C_DIS
LIN {X 59.0818,Y 103.1035,Z 131,A 55.7183,B 24.9399,C -1.79,E1 25.0802,E2 390.3195} C_DIS
LIN {X 61.0989,Y 101.9215,Z 131,A 54.4641,B 24.9405,C -1.7824,E1 25.0832,E2 391.5879} C_DIS
LIN {X 64.2983,Y 99.9339,Z 131,A 52.5538,B 24.9409,C -1.7752,E1 25.0878,E2 393.5092} C_DIS
LIN {X 67.217,Y 97.9943,Z 131,A 50.999,B 24.9407,C -1.7787,E1 25.0914,E2 395.0505} C_DIS
LIN {X 70.0715,Y 95.9738,Z 131,A 49.2144,B 24.9412,C -1.7711,E1 25.0954,E2 396.8466} C_DIS
LIN {X 73.151,Y 93.6483,Z 131,A 47.3094,B 24.9416,C -1.7656,E1 25.0997,E2 398.7576} C_DIS
LIN {X 76.5428,Y 90.897,Z 131,A 45.3194,B 24.9415,C -1.767,E1 25.1039,E2 400.7368} C_DIS
LIN {X 79.3015,Y 88.4994,Z 131,A 43.4695,B 24.942,C -1.7594,E1 25.1078,E2 402.5974} C_DIS
LIN {X 81.9639,Y 86.041,Z 131,A 41.6998,B 24.9423,C -1.7546,E1 25.1114,E2 404.371} C_DIS
LIN {X 85.0895,Y 82.9513,Z 131,A 39.6014,B 24.9425,C -1.751,E1 25.1156,E2 406.4692} C_DIS
LIN {X 88.0503,Y 79.8013,Z 131,A 37.506,B 24.9429,C -1.7458,E1 25.1195,E2 408.5676} C_DIS
LIN {X 90.9246,Y 76.5103,Z 131,A 35.4159,B 24.9432,C -1.7416,E1 25.1233,E2 410.6581} C_DIS
LIN {X 93.6746,Y 73.1176,Z 131,A 33.34,B 24.9434,C -1.7379,E1 25.1269,E2 412.7331} C_DIS
LIN {X 95.6943,Y 70.4539,Z 131,A 31.8978,B 24.9431,C -1.7419,E1 25.1293,E2 414.1589} C_DIS
LIN {X 97.2134,Y 68.3417,Z 131,A 30.6397,B 24.9434,C -1.7385,E1 25.1314,E2 415.4188} C_DIS
LIN {X 98.8081,Y 66.0158,Z 131,A 29.2798,B 24.9436,C -1.735,E1 25.1335,E2 416.7803} C_DIS
LIN {X 100.3938,Y 63.5774,Z 131,A 27.903,B 24.9437,C -1.7325,E1 25.1356,E2 418.156} C_DIS
LIN {X 101.9199,Y 61.1017,Z 131,A 26.4683,B 24.9441,C -1.7272,E1 25.1377,E2 419.596} C_DIS
LIN {X 103.4389,Y 58.4945,Z 131,A 25.0473,B 24.9442,C -1.7248,E1 25.1396,E2 421.0152} C_DIS
LIN {X 105.0237,Y 55.598,Z 131,A 23.5655,B 24.9442,C -1.7257,E1 25.1416,E2 422.4872} C_DIS
LIN {X 106.1893,Y 53.3372,Z 131,A 22.2528,B 24.9447,C -1.7181,E1 25.1433,E2 423.8108} C_DIS
LIN {X 107.4635,Y 50.7228,Z 131,A 20.854,B 24.9449,C -1.7142,E1 25.145,E2 425.2113} C_DIS
LIN {X 108.6717,Y 48.078,Z 131,A 19.4912,B 24.9451,C -1.7121,E1 25.1465,E2 426.5717} C_DIS
LIN {X 109.8156,Y 45.4044,Z 131,A 18.0715,B 24.9454,C -1.7071,E1 25.1481,E2 427.9953} C_DIS
LIN {X 110.8623,Y 42.7866,Z 131,A 16.6781,B 24.9458,C -1.7014,E1 25.1495,E2 429.3944} C_DIS
LIN {X 112.1676,Y 39.235,Z 131,A 14.781,B 24.9463,C -1.6924,E1 25.1513,E2 431.3021} C_DIS
LIN {X 113.3111,Y 35.7999,Z 131,A 13.2124,B 24.9461,C -1.6956,E1 25.1526,E2 432.8542} C_DIS
LIN {X 114.1541,Y 33.0129,Z 131,A 11.7816,B 24.9465,C -1.69,E1 25.1538,E2 434.2901} C_DIS
LIN {X 115.0465,Y 29.7522,Z 131,A 10.0782,B 24.947,C -1.6814,E1 25.155,E2 436.004} C_DIS
LIN {X 115.9475,Y 26.0262,Z 131,A 8.2772,B 24.9472,C -1.6779,E1 25.1562,E2 437.8029} C_DIS
LIN {X 116.5663,Y 23.0941,Z 131,A 6.9285,B 24.9472,C -1.6779,E1 25.1569,E2 439.1435} C_DIS
LIN {X 117.1554,Y 19.8907,Z 131,A 5.4117,B 24.9474,C -1.6756,E1 25.1577,E2 440.6571} C_DIS
LIN {X 117.5633,Y 17.3208,Z 131,A 4.0853,B 24.9479,C -1.6681,E1 25.1582,E2 441.9934} C_DIS
LIN {X 117.9509,Y 14.4444,Z 131,A 2.7041,B 24.9481,C -1.6644,E1 25.1587,E2 443.3749} C_DIS
LIN {X 118.2612,Y 11.6327,Z 131,A 1.3389,B 24.9484,C -1.66,E1 25.1591,E2 444.7426} C_DIS
LIN {X 118.5138,Y 8.6987,Z 131,A -0.118,B 24.9488,C -1.6536,E1 25.1594,E2 446.206} C_DIS
LIN {X 118.6946,Y 5.7162,Z 131,A -1.4633,B 24.9488,C -1.6535,E1 25.1596,E2 447.5435} C_DIS
LIN {X 118.7964,Y 2.9034,Z 131,A -2.8799,B 24.9492,C -1.6462,E1 25.1598,E2 448.9689} C_DIS
LIN {X 118.8326,Y -0.031,Z 131,A -4.2946,B 24.9495,C -1.6415,E1 25.1598,E2 450.3861} C_DIS
LIN {X 118.7937,Y -3.0221,Z 131,A -5.6495,B 24.9495,C -1.6411,E1 25.1598,E2 451.734} C_DIS
LIN {X 118.6885,Y -5.8357,Z 131,A -7.1276,B 24.9502,C -1.6308,E1 25.1595,E2 453.2276} C_DIS
LIN {X 118.5023,Y -8.8489,Z 131,A -8.4982,B 24.9502,C -1.6301,E1 25.1593,E2 454.5916} C_DIS
Enddeposition()
END
